LIN {X 0,Y 320.686,Z 443.971,A -85,B 0,C 180,E1 -15902.996,E2 -15902.996} C_VEL
LIN {X 0,Y 319.386,Z 457.296,A -85,B 0,C 180,E1 -15903.715,E2 -15903.715} C_VEL
LIN {X 0,Y 317.852,Z 469.93,A -85,B 0,C 180,E1 -15904.635,E2 -15904.635} C_VEL
LIN {X 0,Y 316.177,Z 481.923,A -85,B 0,C 180,E1 -15905.756,E2 -15905.756} C_VEL
LIN {X 0,Y 314.275,Z 493.762,A -85,B 0,C 180,E1 -15907.136,E2 -15907.136} C_VEL
LIN {X 0,Y 312.419,Z 503.822,A -85,B 0,C 180,E1 -15908.559,E2 -15908.559} C_VEL
LIN {X 0,Y 310.276,Z 514.883,A -85,B 0,C 180,E1 -15910.483,E2 -15910.483} C_VEL
LIN {X 0,Y 308.49,Z 524.011,A -85,B 0,C 180,E1 -15912.431,E2 -15912.431} C_VEL
LIN {X 0,Y 306.873,Z 532.736,A -85,B 0,C 180,E1 -15914.73,E2 -15914.73} C_VEL
LIN {X 0,Y 305.729,Z 538.879,A -85,B 0,C 180,E1 -15916.711,E2 -15916.711} C_VEL
LIN {X 0,Y 304.809,Z 543.968,A -85,B 0,C 180,E1 -15918.698,E2 -15918.698} C_VEL
LIN {X 0,Y 304.094,Z 549.221,A -85,B 0,C 180,E1 -15921.36,E2 -15921.36} C_VEL
LIN {X 0,Y 303.694,Z 553.281,A -85,B 0,C 180,E1 -15924.322,E2 -15924.322} C_VEL
LIN {X 0,Y 303.583,Z 554.856,A -85,B 0,C 180,E1 -15926.018,E2 -15926.018} C_VEL
LIN {X 0,Y 303.525,Z 556.187,A -85,B 0,C 180,E1 -15928.673,E2 -15928.673} C_VEL
LIN {X 0,Y 303.525,Z 556.181,A -85,B 0,C 180,E1 -15931.327,E2 -15931.327} C_VEL
LIN {X 0,Y 303.584,Z 554.841,A -85,B 0,C 180,E1 -15933.982,E2 -15933.982} C_VEL
LIN {X 0,Y 303.752,Z 552.139,A -85,B 0,C 180,E1 -15936.643,E2 -15936.643} C_VEL
LIN {X 0,Y 304.224,Z 548.001,A -85,B 0,C 180,E1 -15939.306,E2 -15939.306} C_VEL
LIN {X 0,Y 305.041,Z 542.303,A -85,B 0,C 180,E1 -15941.967,E2 -15941.967} C_VEL
LIN {X 0,Y 306.327,Z 535.882,A -85,B 0,C 180,E1 -15944.278,E2 -15944.278} C_VEL
LIN {X 0,Y 307.684,Z 527.905,A -85,B 0,C 180,E1 -15946.589,E2 -15946.589} C_VEL
LIN {X 0,Y 309.31,Z 519.557,A -85,B 0,C 180,E1 -15948.548,E2 -15948.548} C_VEL
LIN {X 0,Y 311.286,Z 509.51,A -85,B 0,C 180,E1 -15950.484,E2 -15950.484} C_VEL
LIN {X 0,Y 313.222,Z 499.398,A -85,B 0,C 180,E1 -15952.075,E2 -15952.075} C_VEL
LIN {X 0,Y 315.371,Z 487.142,A -85,B 0,C 180,E1 -15953.648,E2 -15953.648} C_VEL
LIN {X 0,Y 317.142,Z 474.986,A -85,B 0,C 180,E1 -15954.9,E2 -15954.9} C_VEL
LIN {X 0,Y 318.891,Z 461.491,A -85,B 0,C 180,E1 -15955.977,E2 -15955.977} C_VEL
LIN {X 0,Y 320.356,Z 447.369,A -85,B 0,C 180,E1 -15956.814,E2 -15956.814} C_VEL
LIN {X 0,Y 321.321,Z 433.529,A -85,B 0,C 180,E1 -15957.387,E2 -15957.387} C_VEL
LIN {X 0,Y 322.133,Z 414.857,A -85,B 0,C 180,E1 -15957.841,E2 -15957.841} C_VEL
LIN {X 0,Y 324.269,Z 337.737,A -85,B 0,C 180,E1 -15959.546,E2 -15959.546} C_VEL
LIN {X 0,Y 321.158,Z 321.063,A -85,B 0,C 180,E1 -15960.282,E2 -15960.282} C_VEL
LIN {X 0,Y 313.966,Z 304.498,A -85,B 0,C 180,E1 -15961.482,E2 -15961.482} C_VEL
LIN {X 0,Y 308.979,Z 293.727,A -85,B 0,C 180,E1 -15962.372,E2 -15962.372} C_VEL
LIN {X 0,Y 306.536,Z 284.268,A -85,B 0,C 180,E1 -15965.373,E2 -15965.373} C_VEL
LIN {X 0,Y 305.494,Z 280.07,A -85,B 0,C 180,E1 -15966.89,E2 -15966.89} C_VEL
LIN {X 0,Y 305.452,Z 280.04,A -85,B 0,C 180,E1 -15970.599,E2 -15970.599} C_VEL
LIN {X 0,Y 305.423,Z 280.062,A -85,B 0,C 180,E1 -15973.654,E2 -15973.654} C_VEL
LIN {X 0,Y 305.451,Z 280.062,A -85,B 0,C 180,E1 -15977.414,E2 -15977.414} C_VEL
LIN {X 0,Y 305.491,Z 280.058,A -85,B 0,C 180,E1 -15981.6,E2 -15981.6} C_VEL
LIN {X 0,Y 305.458,Z 280.011,A -85,B 0,C 180,E1 -15984.886,E2 -15984.886} C_VEL
LIN {X 0,Y 305.447,Z 280.048,A -85,B 0,C 180,E1 -15988.354,E2 -15988.354} C_VEL
LIN {X 0,Y 305.516,Z 280.05,A -85,B 0,C 180,E1 -15991.113,E2 -15991.113} C_VEL
LIN {X 0,Y 305.566,Z 280.043,A -85,B 0,C 180,E1 -15994.088,E2 -15994.088} C_VEL
LIN {X 0,Y 305.496,Z 280.042,A -85,B 0,C 180,E1 -15998.403,E2 -15998.403} C_VEL
LIN {X 0,Y 305.585,Z 280.045,A -85,B 0,C 180,E1 -16001.217,E2 -16001.217} C_VEL
LIN {X 0,Y 305.643,Z 280.032,A -85,B 0,C 180,E1 -16005.349,E2 -16005.349} C_VEL
LIN {X 0,Y 305.632,Z 280.02,A -85,B 0,C 180,E1 -16009.4,E2 -16009.4} C_VEL
LIN {X 0,Y 305.807,Z 280.017,A -85,B 0,C 180,E1 -16012.074,E2 -16012.074} C_VEL
LIN {X 0,Y 305.682,Z 280.021,A -85,B 0,C 180,E1 -16014.723,E2 -16014.723} C_VEL
LIN {X 0,Y 305.951,Z 279.997,A -85,B 0,C 180,E1 -16018.684,E2 -16018.684} C_VEL
LIN {X 0,Y 305.951,Z 279.983,A -85,B 0,C 180,E1 -16021.316,E2 -16021.316} C_VEL
LIN {X 0,Y 305.682,Z 280.033,A -85,B 0,C 180,E1 -16025.277,E2 -16025.277} C_VEL
LIN {X 0,Y 305.791,Z 280.004,A -85,B 0,C 180,E1 -16027.926,E2 -16027.926} C_VEL
LIN {X 0,Y 305.597,Z 280.042,A -85,B 0,C 180,E1 -16031.945,E2 -16031.945} C_VEL
LIN {X 0,Y 305.632,Z 280.021,A -85,B 0,C 180,E1 -16035.035,E2 -16035.035} C_VEL
LIN {X 0,Y 305.571,Z 280.038,A -85,B 0,C 180,E1 -16039.445,E2 -16039.445} C_VEL
LIN {X 0,Y 305.486,Z 280.056,A -85,B 0,C 180,E1 -16043.042,E2 -16043.042} C_VEL
LIN {X 0,Y 305.543,Z 280.034,A -85,B 0,C 180,E1 -16046.228,E2 -16046.228} C_VEL
LIN {X 0,Y 305.492,Z 280.058,A -85,B 0,C 180,E1 -16049.051,E2 -16049.051} C_VEL
LIN {X 0,Y 305.461,Z 280.007,A -85,B 0,C 180,E1 -16053.517,E2 -16053.517} C_VEL
LIN {X 0,Y 305.494,Z 280.05,A -85,B 0,C 180,E1 -16056.737,E2 -16056.737} C_VEL
LIN {X 0,Y 305.454,Z 280.025,A -85,B 0,C 180,E1 -16060.601,E2 -16060.601} C_VEL
LIN {X 0,Y 305.417,Z 280.065,A -85,B 0,C 180,E1 -16064.493,E2 -16064.493} C_VEL
LIN {X 0,Y 305.44,Z 280.038,A -85,B 0,C 180,E1 -16068.144,E2 -16068.144} C_VEL
LIN {X 0,Y 305.466,Z 280.045,A -85,B 0,C 180,E1 -16071.597,E2 -16071.597} C_VEL
LIN {X 0,Y 305.522,Z 280.246,A -85,B 0,C 180,E1 -16074.593,E2 -16074.593} C_VEL
LIN {X 0,Y 307.66,Z 288.77,A -85,B 0,C 180,E1 -16077.486,E2 -16077.486} C_VEL
LIN {X 0,Y 310.081,Z 293.827,A -85,B 0,C 180,E1 -16077.97,E2 -16077.97} C_VEL
LIN {X 0,Y 318.342,Z 311.367,A -85,B 0,C 180,E1 -16079.351,E2 -16079.351} C_VEL
LIN {X 0,Y 323.483,Z 324.294,A -85,B 0,C 180,E1 -16080.216,E2 -16080.216} C_VEL
LIN {X 0,Y 324.572,Z 329.961,A -85,B 0,C 180,E1 -16080.467,E2 -16080.467} C_VEL
LIN {X 0,Y 322.075,Z 413.055,A -85,B 0,C 180,E1 -16082.286,E2 -16082.286} C_VEL
LIN {X 0,Y 321.429,Z 429.29,A -85,B 0,C 180,E1 -16082.712,E2 -16082.712} C_VEL
LIN {X 0,Y 320.408,Z 442.749,A -85,B 0,C 180,E1 -16083.279,E2 -16083.279} C_VEL
LIN {X 0,Y 319.032,Z 456.662,A -85,B 0,C 180,E1 -16084.123,E2 -16084.123} C_VEL
LIN {X 0,Y 317.305,Z 470.455,A -85,B 0,C 180,E1 -16085.246,E2 -16085.246} C_VEL
LIN {X 0,Y 315.543,Z 482.714,A -85,B 0,C 180,E1 -16086.54,E2 -16086.54} C_VEL
LIN {X 0,Y 313.618,Z 493.673,A -85,B 0,C 180,E1 -16087.954,E2 -16087.954} C_VEL
LIN {X 0,Y 311.725,Z 503.803,A -85,B 0,C 180,E1 -16089.546,E2 -16089.546} C_VEL
LIN {X 0,Y 309.697,Z 513.859,A -85,B 0,C 180,E1 -16091.476,E2 -16091.476} C_VEL
LIN {X 0,Y 307.923,Z 523.001,A -85,B 0,C 180,E1 -16093.644,E2 -16093.644} C_VEL
LIN {X 0,Y 306.641,Z 530.178,A -85,B 0,C 180,E1 -16095.737,E2 -16095.737} C_VEL
LIN {X 0,Y 305.34,Z 536.596,A -85,B 0,C 180,E1 -16098.045,E2 -16098.045} C_VEL
LIN {X 0,Y 304.429,Z 542.285,A -85,B 0,C 180,E1 -16100.7,E2 -16100.7} C_VEL
LIN {X 0,Y 303.921,Z 546.419,A -85,B 0,C 180,E1 -16103.361,E2 -16103.361} C_VEL
LIN {X 0,Y 303.673,Z 549.122,A -85,B 0,C 180,E1 -16106.019,E2 -16106.019} C_VEL
LIN {X 0,Y 303.538,Z 550.476,A -85,B 0,C 180,E1 -16108.673,E2 -16108.673} C_VEL
LIN {X 0,Y 303.538,Z 550.507,A -85,B 0,C 180,E1 -16111.327,E2 -16111.327} C_VEL
LIN {X 0,Y 303.673,Z 549.213,A -85,B 0,C 180,E1 -16113.981,E2 -16113.981} C_VEL
LIN {X 0,Y 303.92,Z 546.564,A -85,B 0,C 180,E1 -16116.639,E2 -16116.639} C_VEL
LIN {X 0,Y 304.418,Z 542.492,A -85,B 0,C 180,E1 -16119.3,E2 -16119.3} C_VEL
LIN {X 0,Y 305.314,Z 536.866,A -85,B 0,C 180,E1 -16121.956,E2 -16121.956} C_VEL
LIN {X 0,Y 306.586,Z 530.512,A -85,B 0,C 180,E1 -16124.266,E2 -16124.266} C_VEL
LIN {X 0,Y 308.067,Z 522.382,A -85,B 0,C 180,E1 -16126.633,E2 -16126.633} C_VEL
LIN {X 0,Y 309.653,Z 514.35,A -85,B 0,C 180,E1 -16128.526,E2 -16128.526} C_VEL
LIN {X 0,Y 311.6,Z 504.392,A -85,B 0,C 180,E1 -16130.462,E2 -16130.462} C_VEL
LIN {X 0,Y 313.732,Z 493.305,A -85,B 0,C 180,E1 -16132.211,E2 -16132.211} C_VEL
LIN {X 0,Y 315.655,Z 482.266,A -85,B 0,C 180,E1 -16133.625,E2 -16133.625} C_VEL
LIN {X 0,Y 317.426,Z 470.279,A -85,B 0,C 180,E1 -16134.876,E2 -16134.876} C_VEL
LIN {X 0,Y 319.064,Z 457.023,A -85,B 0,C 180,E1 -16135.962,E2 -16135.962} C_VEL
LIN {X 0,Y 320.387,Z 443.995,A -85,B 0,C 180,E1 -16136.767,E2 -16136.767} C_VEL
LIN {X 0,Y 321.438,Z 429.999,A -85,B 0,C 180,E1 -16137.375,E2 -16137.375} C_VEL
LIN {X 0,Y 322.139,Z 412.365,A -85,B 0,C 180,E1 -16137.84,E2 -16137.84} C_VEL
LIN {X 0,Y 324.009,Z 350.719,A -85,B 0,C 180,E1 -16139.188,E2 -16139.188} C_VEL
LIN {X 0,Y 324.421,Z 329.108,A -85,B 0,C 180,E1 -16139.685,E2 -16139.685} C_VEL
LIN {X 0,Y 323.131,Z 323.106,A -85,B 0,C 180,E1 -16139.967,E2 -16139.967} C_VEL
LIN {X 0,Y 315.3,Z 304.632,A -85,B 0,C 180,E1 -16141.273,E2 -16141.273} C_VEL
LIN {X 0,Y 307.781,Z 289.059,A -85,B 0,C 180,E1 -16142.584,E2 -16142.584} C_VEL
LIN {X 0,Y 306.579,Z 284.524,A -85,B 0,C 180,E1 -16144.015,E2 -16144.015} C_VEL
LIN {X 0,Y 306.149,Z 282.788,A -85,B 0,C 180,E1 -16144.61,E2 -16144.61} C_VEL
LIN {X 0,Y 305.43,Z 281.38,A -85,B 0,C 180,E1 -16145.27,E2 -16145.27} C_VEL
LIN {X 0,Y 303.733,Z 280.518,A -85,B 0,C 180,E1 -16146.312,E2 -16146.312} C_VEL
LIN {X 0,Y 299.402,Z 280.805,A -85,B 0,C 180,E1 -16148.856,E2 -16148.856} C_VEL
LIN {X 0,Y 298.436,Z 280.938,A -85,B 0,C 180,E1 -16150.005,E2 -16150.005} C_VEL
LIN {X 0,Y 298.362,Z 280.932,A -85,B 0,C 180,E1 -16150.393,E2 -16150.393} C_VEL
LIN {X 0,Y 298.396,Z 280.916,A -85,B 0,C 180,E1 -16153.102,E2 -16153.102} C_VEL
LIN {X 0,Y 298.4,Z 280.916,A -85,B 0,C 180,E1 -16156.92,E2 -16156.92} C_VEL
LIN {X 0,Y 298.418,Z 280.931,A -85,B 0,C 180,E1 -16161.001,E2 -16161.001} C_VEL
LIN {X 0,Y 298.427,Z 280.925,A -85,B 0,C 180,E1 -16163.931,E2 -16163.931} C_VEL
LIN {X 0,Y 298.39,Z 280.899,A -85,B 0,C 180,E1 -16167.983,E2 -16167.983} C_VEL
LIN {X 0,Y 298.459,Z 280.933,A -85,B 0,C 180,E1 -16171.904,E2 -16171.904} C_VEL
LIN {X 0,Y 298.48,Z 280.92,A -85,B 0,C 180,E1 -16174.923,E2 -16174.923} C_VEL
LIN {X 0,Y 298.444,Z 280.918,A -85,B 0,C 180,E1 -16179.315,E2 -16179.315} C_VEL
LIN {X 0,Y 298.532,Z 280.923,A -85,B 0,C 180,E1 -16182.179,E2 -16182.179} C_VEL
LIN {X 0,Y 298.587,Z 280.898,A -85,B 0,C 180,E1 -16184.994,E2 -16184.994} C_VEL
LIN {X 0,Y 298.585,Z 280.911,A -85,B 0,C 180,E1 -16189.146,E2 -16189.146} C_VEL
LIN {X 0,Y 298.735,Z 280.88,A -85,B 0,C 180,E1 -16191.885,E2 -16191.885} C_VEL
LIN {X 0,Y 298.652,Z 280.91,A -85,B 0,C 180,E1 -16194.599,E2 -16194.599} C_VEL
LIN {X 0,Y 298.918,Z 280.858,A -85,B 0,C 180,E1 -16198.653,E2 -16198.653} C_VEL
LIN {X 0,Y 298.918,Z 280.873,A -85,B 0,C 180,E1 -16201.347,E2 -16201.347} C_VEL
LIN {X 0,Y 298.791,Z 280.892,A -85,B 0,C 180,E1 -16206.754,E2 -16206.754} C_VEL
LIN {X 0,Y 298.674,Z 280.89,A -85,B 0,C 180,E1 -16209.481,E2 -16209.481} C_VEL
LIN {X 0,Y 298.545,Z 280.922,A -85,B 0,C 180,E1 -16213.616,E2 -16213.616} C_VEL
LIN {X 0,Y 298.542,Z 280.904,A -85,B 0,C 180,E1 -16216.409,E2 -16216.409} C_VEL
LIN {X 0,Y 298.506,Z 280.927,A -85,B 0,C 180,E1 -16219.655,E2 -16219.655} C_VEL
LIN {X 0,Y 298.452,Z 280.927,A -85,B 0,C 180,E1 -16223.598,E2 -16223.598} C_VEL
LIN {X 0,Y 298.484,Z 280.918,A -85,B 0,C 180,E1 -16226.575,E2 -16226.575} C_VEL
LIN {X 0,Y 298.416,Z 280.938,A -85,B 0,C 180,E1 -16229.641,E2 -16229.641} C_VEL
LIN {X 0,Y 298.39,Z 280.903,A -85,B 0,C 180,E1 -16232.801,E2 -16232.801} C_VEL
LIN {X 0,Y 298.442,Z 280.913,A -85,B 0,C 180,E1 -16236.808,E2 -16236.808} C_VEL
LIN {X 0,Y 298.404,Z 280.935,A -85,B 0,C 180,E1 -16239.487,E2 -16239.487} C_VEL
LIN {X 0,Y 298.422,Z 280.935,A -85,B 0,C 180,E1 -16243.11,E2 -16243.11} C_VEL
LIN {X 0,Y 298.464,Z 280.915,A -85,B 0,C 180,E1 -16246.933,E2 -16246.933} C_VEL
LIN {X 0,Y 298.431,Z 280.937,A -85,B 0,C 180,E1 -16251,E2 -16251} C_VEL
LIN {X 0,Y 298.481,Z 280.971,A -85,B 0,C 180,E1 -16252.384,E2 -16252.384} C_VEL
LIN {X 0,Y 301.015,Z 291,A -85,B 0,C 180,E1 -16255.921,E2 -16255.921} C_VEL
LIN {X 0,Y 301.722,Z 293.772,A -85,B 0,C 180,E1 -16256.725,E2 -16256.725} C_VEL
LIN {X 0,Y 310.639,Z 312.674,A -85,B 0,C 180,E1 -16258.33,E2 -16258.33} C_VEL
LIN {X 0,Y 315.731,Z 325.016,A -85,B 0,C 180,E1 -16259.217,E2 -16259.217} C_VEL
LIN {X 0,Y 318.186,Z 339.496,A -85,B 0,C 180,E1 -16259.851,E2 -16259.851} C_VEL
LIN {X 0,Y 315.386,Z 429.211,A -85,B 0,C 180,E1 -16261.873,E2 -16261.873} C_VEL
LIN {X 0,Y 314.376,Z 443.915,A -85,B 0,C 180,E1 -16262.409,E2 -16262.409} C_VEL
LIN {X 0,Y 313.05,Z 457.237,A -85,B 0,C 180,E1 -16263.141,E2 -16263.141} C_VEL
LIN {X 0,Y 311.442,Z 469.869,A -85,B 0,C 180,E1 -16264.074,E2 -16264.074} C_VEL
LIN {X 0,Y 309.639,Z 482.266,A -85,B 0,C 180,E1 -16265.26,E2 -16265.26} C_VEL
LIN {X 0,Y 307.497,Z 494.874,A -85,B 0,C 180,E1 -16266.781,E2 -16266.781} C_VEL
LIN {X 0,Y 305.352,Z 505.724,A -85,B 0,C 180,E1 -16268.392,E2 -16268.392} C_VEL
LIN {X 0,Y 303.216,Z 516.448,A -85,B 0,C 180,E1 -16270.362,E2 -16270.362} C_VEL
LIN {X 0,Y 301.404,Z 525.302,A -85,B 0,C 180,E1 -16272.355,E2 -16272.355} C_VEL
LIN {X 0,Y 299.755,Z 533.789,A -85,B 0,C 180,E1 -16274.707,E2 -16274.707} C_VEL
LIN {X 0,Y 298.419,Z 540.627,A -85,B 0,C 180,E1 -16277.072,E2 -16277.072} C_VEL
LIN {X 0,Y 297.591,Z 545.338,A -85,B 0,C 180,E1 -16279.11,E2 -16279.11} C_VEL
LIN {X 0,Y 296.91,Z 550.222,A -85,B 0,C 180,E1 -16281.835,E2 -16281.835} C_VEL
LIN {X 0,Y 296.553,Z 553.616,A -85,B 0,C 180,E1 -16284.561,E2 -16284.561} C_VEL
LIN {X 0,Y 296.481,Z 555.623,A -85,B 0,C 180,E1 -16287.283,E2 -16287.283} C_VEL
LIN {X 0,Y 296.45,Z 556.284,A -85,B 0,C 180,E1 -16290,E2 -16290} C_VEL
LIN {X 0,Y 296.481,Z 555.612,A -85,B 0,C 180,E1 -16292.717,E2 -16292.717} C_VEL
LIN {X 0,Y 296.587,Z 553.433,A -85,B 0,C 180,E1 -16295.592,E2 -16295.592} C_VEL
LIN {X 0,Y 296.91,Z 550.189,A -85,B 0,C 180,E1 -16298.165,E2 -16298.165} C_VEL
LIN {X 0,Y 297.593,Z 545.288,A -85,B 0,C 180,E1 -16300.89,E2 -16300.89} C_VEL
LIN {X 0,Y 298.419,Z 540.563,A -85,B 0,C 180,E1 -16302.928,E2 -16302.928} C_VEL
LIN {X 0,Y 299.732,Z 533.725,A -85,B 0,C 180,E1 -16305.29,E2 -16305.29} C_VEL
LIN {X 0,Y 301.113,Z 526.564,A -85,B 0,C 180,E1 -16307.312,E2 -16307.312} C_VEL
LIN {X 0,Y 302.891,Z 517.962,A -85,B 0,C 180,E1 -16309.307,E2 -16309.307} C_VEL
LIN {X 0,Y 304.954,Z 507.536,A -85,B 0,C 180,E1 -16311.283,E2 -16311.283} C_VEL
LIN {X 0,Y 307.098,Z 497.053,A -85,B 0,C 180,E1 -16312.895,E2 -16312.895} C_VEL
LIN {X 0,Y 309.239,Z 484.476,A -85,B 0,C 180,E1 -16314.472,E2 -16314.472} C_VEL
LIN {X 0,Y 311.205,Z 471.378,A -85,B 0,C 180,E1 -16315.767,E2 -16315.767} C_VEL
LIN {X 0,Y 312.923,Z 458.027,A -85,B 0,C 180,E1 -16316.781,E2 -16316.781} C_VEL
LIN {X 0,Y 314.294,Z 444.238,A -85,B 0,C 180,E1 -16317.554,E2 -16317.554} C_VEL
LIN {X 0,Y 315.369,Z 429.817,A -85,B 0,C 180,E1 -16318.084,E2 -16318.084} C_VEL
LIN {X 0,Y 318.117,Z 339.637,A -85,B 0,C 180,E1 -16320.125,E2 -16320.125} C_VEL
LIN {X 0,Y 315.49,Z 324.243,A -85,B 0,C 180,E1 -16320.8,E2 -16320.8} C_VEL
LIN {X 0,Y 308.305,Z 307.631,A -85,B 0,C 180,E1 -16322.042,E2 -16322.042} C_VEL
LIN {X 0,Y 301.672,Z 293.605,A -85,B 0,C 180,E1 -16323.26,E2 -16323.26} C_VEL
LIN {X 0,Y 299.336,Z 284.508,A -85,B 0,C 180,E1 -16326.258,E2 -16326.258} C_VEL
LIN {X 0,Y 298.44,Z 280.947,A -85,B 0,C 180,E1 -16327.621,E2 -16327.621} C_VEL
LIN {X 0,Y 298.381,Z 280.915,A -85,B 0,C 180,E1 -16331.261,E2 -16331.261} C_VEL
LIN {X 0,Y 298.351,Z 280.943,A -85,B 0,C 180,E1 -16335.034,E2 -16335.034} C_VEL
LIN {X 0,Y 298.38,Z 280.934,A -85,B 0,C 180,E1 -16338.738,E2 -16338.738} C_VEL
LIN {X 0,Y 298.421,Z 280.932,A -85,B 0,C 180,E1 -16342.243,E2 -16342.243} C_VEL
LIN {X 0,Y 298.403,Z 280.887,A -85,B 0,C 180,E1 -16345.581,E2 -16345.581} C_VEL
LIN {X 0,Y 298.391,Z 280.934,A -85,B 0,C 180,E1 -16348.791,E2 -16348.791} C_VEL
LIN {X 0,Y 298.459,Z 280.92,A -85,B 0,C 180,E1 -16351.904,E2 -16351.904} C_VEL
LIN {X 0,Y 298.481,Z 280.929,A -85,B 0,C 180,E1 -16354.924,E2 -16354.924} C_VEL
LIN {X 0,Y 298.445,Z 280.928,A -85,B 0,C 180,E1 -16359.315,E2 -16359.315} C_VEL
LIN {X 0,Y 298.532,Z 280.913,A -85,B 0,C 180,E1 -16362.179,E2 -16362.179} C_VEL
LIN {X 0,Y 298.588,Z 280.909,A -85,B 0,C 180,E1 -16364.995,E2 -16364.995} C_VEL
LIN {X 0,Y 298.587,Z 280.898,A -85,B 0,C 180,E1 -16369.146,E2 -16369.146} C_VEL
LIN {X 0,Y 298.753,Z 280.893,A -85,B 0,C 180,E1 -16371.886,E2 -16371.886} C_VEL
LIN {X 0,Y 298.654,Z 280.898,A -85,B 0,C 180,E1 -16374.599,E2 -16374.599} C_VEL
LIN {X 0,Y 298.917,Z 280.873,A -85,B 0,C 180,E1 -16378.653,E2 -16378.653} C_VEL
LIN {X 0,Y 298.918,Z 280.859,A -85,B 0,C 180,E1 -16381.347,E2 -16381.347} C_VEL
LIN {X 0,Y 298.782,Z 280.89,A -85,B 0,C 180,E1 -16386.754,E2 -16386.754} C_VEL
LIN {X 0,Y 298.63,Z 280.893,A -85,B 0,C 180,E1 -16389.482,E2 -16389.482} C_VEL
LIN {X 0,Y 298.546,Z 280.911,A -85,B 0,C 180,E1 -16393.616,E2 -16393.616} C_VEL
LIN {X 0,Y 298.543,Z 280.914,A -85,B 0,C 180,E1 -16396.409,E2 -16396.409} C_VEL
LIN {X 0,Y 298.506,Z 280.917,A -85,B 0,C 180,E1 -16399.655,E2 -16399.655} C_VEL
LIN {X 0,Y 298.453,Z 280.934,A -85,B 0,C 180,E1 -16403.598,E2 -16403.598} C_VEL
LIN {X 0,Y 298.485,Z 280.914,A -85,B 0,C 180,E1 -16406.575,E2 -16406.575} C_VEL
LIN {X 0,Y 298.417,Z 280.935,A -85,B 0,C 180,E1 -16409.642,E2 -16409.642} C_VEL
LIN {X 0,Y 298.391,Z 280.889,A -85,B 0,C 180,E1 -16412.801,E2 -16412.801} C_VEL
LIN {X 0,Y 298.462,Z 280.926,A -85,B 0,C 180,E1 -16416.813,E2 -16416.813} C_VEL
LIN {X 0,Y 298.411,Z 280.92,A -85,B 0,C 180,E1 -16419.486,E2 -16419.486} C_VEL
LIN {X 0,Y 298.396,Z 280.913,A -85,B 0,C 180,E1 -16423.104,E2 -16423.104} C_VEL
LIN {X 0,Y 298.401,Z 280.916,A -85,B 0,C 180,E1 -16426.921,E2 -16426.921} C_VEL
LIN {X 0,Y 298.397,Z 280.932,A -85,B 0,C 180,E1 -16431.008,E2 -16431.008} C_VEL
LIN {X 0,Y 298.464,Z 281.067,A -85,B 0,C 180,E1 -16433.845,E2 -16433.845} C_VEL
LIN {X 0,Y 300.51,Z 288.901,A -85,B 0,C 180,E1 -16436.622,E2 -16436.622} C_VEL
LIN {X 0,Y 303.356,Z 294.889,A -85,B 0,C 180,E1 -16437.198,E2 -16437.198} C_VEL
LIN {X 0,Y 311.058,Z 310.831,A -85,B 0,C 180,E1 -16438.535,E2 -16438.535} C_VEL
LIN {X 0,Y 317.44,Z 326.268,A -85,B 0,C 180,E1 -16439.638,E2 -16439.638} C_VEL
LIN {X 0,Y 318.353,Z 331.68,A -85,B 0,C 180,E1 -16439.873,E2 -16439.873} C_VEL
LIN {X 0,Y 315.887,Z 411.357,A -85,B 0,C 180,E1 -16441.65,E2 -16441.65} C_VEL
LIN {X 0,Y 315.155,Z 429.372,A -85,B 0,C 180,E1 -16442.122,E2 -16442.122} C_VEL
LIN {X 0,Y 314.028,Z 443.587,A -85,B 0,C 180,E1 -16442.736,E2 -16442.736} C_VEL
LIN {X 0,Y 312.642,Z 456.736,A -85,B 0,C 180,E1 -16443.553,E2 -16443.553} C_VEL
LIN {X 0,Y 310.879,Z 470.492,A -85,B 0,C 180,E1 -16444.695,E2 -16444.695} C_VEL
LIN {X 0,Y 309.042,Z 482.785,A -85,B 0,C 180,E1 -16446.015,E2 -16446.015} C_VEL
LIN {X 0,Y 306.824,Z 494.811,A -85,B 0,C 180,E1 -16447.617,E2 -16447.617} C_VEL
LIN {X 0,Y 304.695,Z 505.652,A -85,B 0,C 180,E1 -16449.406,E2 -16449.406} C_VEL
LIN {X 0,Y 302.639,Z 515.411,A -85,B 0,C 180,E1 -16451.379,E2 -16451.379} C_VEL
LIN {X 0,Y 300.993,Z 523.541,A -85,B 0,C 180,E1 -16453.391,E2 -16453.391} C_VEL
LIN {X 0,Y 299.753,Z 530.246,A -85,B 0,C 180,E1 -16455.402,E2 -16455.402} C_VEL
LIN {X 0,Y 298.355,Z 536.664,A -85,B 0,C 180,E1 -16457.76,E2 -16457.76} C_VEL
LIN {X 0,Y 297.39,Z 542.353,A -85,B 0,C 180,E1 -16460.478,E2 -16460.478} C_VEL
LIN {X 0,Y 296.854,Z 546.486,A -85,B 0,C 180,E1 -16463.202,E2 -16463.202} C_VEL
LIN {X 0,Y 296.575,Z 549.189,A -85,B 0,C 180,E1 -16465.923,E2 -16465.923} C_VEL
LIN {X 0,Y 296.46,Z 550.542,A -85,B 0,C 180,E1 -16468.642,E2 -16468.642} C_VEL
LIN {X 0,Y 296.459,Z 550.573,A -85,B 0,C 180,E1 -16471.358,E2 -16471.358} C_VEL
LIN {X 0,Y 296.575,Z 549.279,A -85,B 0,C 180,E1 -16474.077,E2 -16474.077} C_VEL
LIN {X 0,Y 296.854,Z 546.63,A -85,B 0,C 180,E1 -16476.798,E2 -16476.798} C_VEL
LIN {X 0,Y 297.377,Z 542.557,A -85,B 0,C 180,E1 -16479.522,E2 -16479.522} C_VEL
LIN {X 0,Y 298.329,Z 536.932,A -85,B 0,C 180,E1 -16482.24,E2 -16482.24} C_VEL
LIN {X 0,Y 299.696,Z 530.577,A -85,B 0,C 180,E1 -16484.601,E2 -16484.601} C_VEL
LIN {X 0,Y 301.114,Z 522.987,A -85,B 0,C 180,E1 -16486.875,E2 -16486.875} C_VEL
LIN {X 0,Y 302.893,Z 514.414,A -85,B 0,C 180,E1 -16488.955,E2 -16488.955} C_VEL
LIN {X 0,Y 304.93,Z 504.456,A -85,B 0,C 180,E1 -16490.93,E2 -16490.93} C_VEL
LIN {X 0,Y 307.17,Z 493.368,A -85,B 0,C 180,E1 -16492.711,E2 -16492.711} C_VEL
LIN {X 0,Y 309.171,Z 482.327,A -85,B 0,C 180,E1 -16494.152,E2 -16494.152} C_VEL
LIN {X 0,Y 310.976,Z 470.34,A -85,B 0,C 180,E1 -16495.429,E2 -16495.429} C_VEL
LIN {X 0,Y 312.701,Z 457.082,A -85,B 0,C 180,E1 -16496.531,E2 -16496.531} C_VEL
LIN {X 0,Y 314.07,Z 444.051,A -85,B 0,C 180,E1 -16497.35,E2 -16497.35} C_VEL
LIN {X 0,Y 315.166,Z 430.049,A -85,B 0,C 180,E1 -16497.968,E2 -16497.968} C_VEL
LIN {X 0,Y 315.894,Z 412.407,A -85,B 0,C 180,E1 -16498.44,E2 -16498.44} C_VEL
LIN {X 0,Y 317.784,Z 353.431,A -85,B 0,C 180,E1 -16499.748,E2 -16499.748} C_VEL
LIN {X 0,Y 318.334,Z 330.709,A -85,B 0,C 180,E1 -16500.272,E2 -16500.272} C_VEL
LIN {X 0,Y 317.386,Z 326.064,A -85,B 0,C 180,E1 -16500.491,E2 -16500.491} C_VEL
LIN {X 0,Y 309.604,Z 307.643,A -85,B 0,C 180,E1 -16501.836,E2 -16501.836} C_VEL
LIN {X 0,Y 302.014,Z 292.202,A -85,B 0,C 180,E1 -16503.165,E2 -16503.165} C_VEL
LIN {X 0,Y 300.432,Z 288.707,A -85,B 0,C 180,E1 -16503.545,E2 -16503.545} C_VEL
LIN {X 0,Y 298.47,Z 281.117,A -85,B 0,C 180,E1 -16506.246,E2 -16506.246} C_VEL
LIN {X 0,Y 298.399,Z 280.939,A -85,B 0,C 180,E1 -16509.487,E2 -16509.487} C_VEL
LIN {X 0,Y 298.362,Z 280.932,A -85,B 0,C 180,E1 -16510.393,E2 -16510.393} C_VEL
LIN {X 0,Y 297.71,Z 281.012,A -85,B 0,C 180,E1 -16511.52,E2 -16511.52} C_VEL
LIN {X 0,Y 294.888,Z 281.378,A -85,B 0,C 180,E1 -16513.356,E2 -16513.356} C_VEL
LIN {X 0,Y 292.472,Z 281.684,A -85,B 0,C 180,E1 -16514.845,E2 -16514.845} C_VEL
LIN {X 0,Y 291.413,Z 281.805,A -85,B 0,C 180,E1 -16515.999,E2 -16515.999} C_VEL
LIN {X 0,Y 291.315,Z 281.808,A -85,B 0,C 180,E1 -16516.39,E2 -16516.39} C_VEL
LIN {X 0,Y 291.388,Z 281.793,A -85,B 0,C 180,E1 -16520.515,E2 -16520.515} C_VEL
LIN {X 0,Y 291.422,Z 281.812,A -85,B 0,C 180,E1 -16522.922,E2 -16522.922} C_VEL
LIN {X 0,Y 291.34,Z 281.768,A -85,B 0,C 180,E1 -16526.301,E2 -16526.301} C_VEL
LIN {X 0,Y 291.383,Z 281.812,A -85,B 0,C 180,E1 -16530.259,E2 -16530.259} C_VEL
LIN {X 0,Y 291.411,Z 281.795,A -85,B 0,C 180,E1 -16534.271,E2 -16534.271} C_VEL
LIN {X 0,Y 291.376,Z 281.812,A -85,B 0,C 180,E1 -16537.299,E2 -16537.299} C_VEL
LIN {X 0,Y 291.453,Z 281.794,A -85,B 0,C 180,E1 -16540.27,E2 -16540.27} C_VEL
LIN {X 0,Y 291.535,Z 281.777,A -85,B 0,C 180,E1 -16544.634,E2 -16544.634} C_VEL
LIN {X 0,Y 291.529,Z 281.792,A -85,B 0,C 180,E1 -16548.88,E2 -16548.88} C_VEL
LIN {X 0,Y 291.681,Z 281.757,A -85,B 0,C 180,E1 -16551.688,E2 -16551.688} C_VEL
LIN {X 0,Y 291.622,Z 281.786,A -85,B 0,C 180,E1 -16554.468,E2 -16554.468} C_VEL
LIN {X 0,Y 291.884,Z 281.733,A -85,B 0,C 180,E1 -16558.62,E2 -16558.62} C_VEL
LIN {X 0,Y 291.884,Z 281.749,A -85,B 0,C 180,E1 -16561.38,E2 -16561.38} C_VEL
LIN {X 0,Y 291.739,Z 281.769,A -85,B 0,C 180,E1 -16566.918,E2 -16566.918} C_VEL
LIN {X 0,Y 291.623,Z 281.766,A -85,B 0,C 180,E1 -16569.712,E2 -16569.712} C_VEL
LIN {X 0,Y 291.515,Z 281.799,A -85,B 0,C 180,E1 -16573.951,E2 -16573.951} C_VEL
LIN {X 0,Y 291.481,Z 281.784,A -85,B 0,C 180,E1 -16576.818,E2 -16576.818} C_VEL
LIN {X 0,Y 291.445,Z 281.807,A -85,B 0,C 180,E1 -16579.875,E2 -16579.875} C_VEL
LIN {X 0,Y 291.395,Z 281.811,A -85,B 0,C 180,E1 -16584.206,E2 -16584.206} C_VEL
LIN {X 0,Y 291.417,Z 281.795,A -85,B 0,C 180,E1 -16587.272,E2 -16587.272} C_VEL
LIN {X 0,Y 291.333,Z 281.819,A -85,B 0,C 180,E1 -16590.437,E2 -16590.437} C_VEL
LIN {X 0,Y 291.339,Z 281.769,A -85,B 0,C 180,E1 -16593.699,E2 -16593.699} C_VEL
LIN {X 0,Y 291.377,Z 281.803,A -85,B 0,C 180,E1 -16597.256,E2 -16597.256} C_VEL
LIN {X 0,Y 291.333,Z 281.809,A -85,B 0,C 180,E1 -16600.642,E2 -16600.642} C_VEL
LIN {X 0,Y 291.338,Z 281.813,A -85,B 0,C 180,E1 -16604.393,E2 -16604.393} C_VEL
LIN {X 0,Y 291.385,Z 281.785,A -85,B 0,C 180,E1 -16608.391,E2 -16608.391} C_VEL
LIN {X 0,Y 291.425,Z 281.927,A -85,B 0,C 180,E1 -16611.68,E2 -16611.68} C_VEL
LIN {X 0,Y 293.777,Z 290.926,A -85,B 0,C 180,E1 -16614.961,E2 -16614.961} C_VEL
LIN {X 0,Y 294.451,Z 293.564,A -85,B 0,C 180,E1 -16615.781,E2 -16615.781} C_VEL
LIN {X 0,Y 303.669,Z 312.839,A -85,B 0,C 180,E1 -16617.521,E2 -16617.521} C_VEL
LIN {X 0,Y 309.857,Z 327.379,A -85,B 0,C 180,E1 -16618.632,E2 -16618.632} C_VEL
LIN {X 0,Y 312.063,Z 340.503,A -85,B 0,C 180,E1 -16619.223,E2 -16619.223} C_VEL
LIN {X 0,Y 309.158,Z 429.163,A -85,B 0,C 180,E1 -16621.254,E2 -16621.254} C_VEL
LIN {X 0,Y 308.114,Z 443.858,A -85,B 0,C 180,E1 -16621.798,E2 -16621.798} C_VEL
LIN {X 0,Y 306.742,Z 457.177,A -85,B 0,C 180,E1 -16622.543,E2 -16622.543} C_VEL
LIN {X 0,Y 305.071,Z 469.808,A -85,B 0,C 180,E1 -16623.491,E2 -16623.491} C_VEL
LIN {X 0,Y 303.061,Z 482.921,A -85,B 0,C 180,E1 -16624.778,E2 -16624.778} C_VEL
LIN {X 0,Y 300.963,Z 494.81,A -85,B 0,C 180,E1 -16626.246,E2 -16626.246} C_VEL
LIN {X 0,Y 298.74,Z 505.66,A -85,B 0,C 180,E1 -16627.889,E2 -16627.889} C_VEL
LIN {X 0,Y 296.498,Z 516.383,A -85,B 0,C 180,E1 -16629.898,E2 -16629.898} C_VEL
LIN {X 0,Y 294.609,Z 525.237,A -85,B 0,C 180,E1 -16631.934,E2 -16631.934} C_VEL
LIN {X 0,Y 292.888,Z 533.723,A -85,B 0,C 180,E1 -16634.339,E2 -16634.339} C_VEL
LIN {X 0,Y 291.476,Z 540.561,A -85,B 0,C 180,E1 -16636.759,E2 -16636.759} C_VEL
LIN {X 0,Y 290.578,Z 545.272,A -85,B 0,C 180,E1 -16638.844,E2 -16638.844} C_VEL
LIN {X 0,Y 289.86,Z 550.156,A -85,B 0,C 180,E1 -16641.635,E2 -16641.635} C_VEL
LIN {X 0,Y 289.471,Z 553.646,A -85,B 0,C 180,E1 -16644.519,E2 -16644.519} C_VEL
LIN {X 0,Y 289.388,Z 555.557,A -85,B 0,C 180,E1 -16647.216,E2 -16647.216} C_VEL
LIN {X 0,Y 289.37,Z 556.218,A -85,B 0,C 180,E1 -16650,E2 -16650} C_VEL
LIN {X 0,Y 289.388,Z 555.545,A -85,B 0,C 180,E1 -16652.784,E2 -16652.784} C_VEL
LIN {X 0,Y 289.48,Z 553.529,A -85,B 0,C 180,E1 -16655.573,E2 -16655.573} C_VEL
LIN {X 0,Y 289.86,Z 550.121,A -85,B 0,C 180,E1 -16658.365,E2 -16658.365} C_VEL
LIN {X 0,Y 290.58,Z 545.22,A -85,B 0,C 180,E1 -16661.156,E2 -16661.156} C_VEL
LIN {X 0,Y 291.476,Z 540.495,A -85,B 0,C 180,E1 -16663.242,E2 -16663.242} C_VEL
LIN {X 0,Y 292.851,Z 533.672,A -85,B 0,C 180,E1 -16665.654,E2 -16665.654} C_VEL
LIN {X 0,Y 294.298,Z 526.494,A -85,B 0,C 180,E1 -16667.726,E2 -16667.726} C_VEL
LIN {X 0,Y 296.169,Z 517.892,A -85,B 0,C 180,E1 -16669.764,E2 -16669.764} C_VEL
LIN {X 0,Y 298.32,Z 507.466,A -85,B 0,C 180,E1 -16671.78,E2 -16671.78} C_VEL
LIN {X 0,Y 300.563,Z 496.983,A -85,B 0,C 180,E1 -16673.422,E2 -16673.422} C_VEL
LIN {X 0,Y 302.752,Z 484.405,A -85,B 0,C 180,E1 -16675.031,E2 -16675.031} C_VEL
LIN {X 0,Y 304.817,Z 471.306,A -85,B 0,C 180,E1 -16676.348,E2 -16676.348} C_VEL
LIN {X 0,Y 306.587,Z 457.954,A -85,B 0,C 180,E1 -16677.38,E2 -16677.38} C_VEL
LIN {X 0,Y 308.022,Z 444.162,A -85,B 0,C 180,E1 -16678.165,E2 -16678.165} C_VEL
LIN {X 0,Y 309.124,Z 429.733,A -85,B 0,C 180,E1 -16678.703,E2 -16678.703} C_VEL
LIN {X 0,Y 311.924,Z 342.841,A -85,B 0,C 180,E1 -16680.701,E2 -16680.701} C_VEL
LIN {X 0,Y 311.599,Z 338.261,A -85,B 0,C 180,E1 -16680.857,E2 -16680.857} C_VEL
LIN {X 0,Y 309.484,Z 326.458,A -85,B 0,C 180,E1 -16681.404,E2 -16681.404} C_VEL
LIN {X 0,Y 301.76,Z 308.636,A -85,B 0,C 180,E1 -16682.793,E2 -16682.793} C_VEL
LIN {X 0,Y 295.598,Z 296.169,A -85,B 0,C 180,E1 -16683.92,E2 -16683.92} C_VEL
LIN {X 0,Y 294.347,Z 293.248,A -85,B 0,C 180,E1 -16684.25,E2 -16684.25} C_VEL
LIN {X 0,Y 291.989,Z 284.154,A -85,B 0,C 180,E1 -16687.412,E2 -16687.412} C_VEL
LIN {X 0,Y 291.363,Z 281.836,A -85,B 0,C 180,E1 -16688.376,E2 -16688.376} C_VEL
LIN {X 0,Y 291.316,Z 281.798,A -85,B 0,C 180,E1 -16692.492,E2 -16692.492} C_VEL
LIN {X 0,Y 291.306,Z 281.817,A -85,B 0,C 180,E1 -16696.366,E2 -16696.366} C_VEL
LIN {X 0,Y 291.383,Z 281.81,A -85,B 0,C 180,E1 -16700.516,E2 -16700.516} C_VEL
LIN {X 0,Y 291.407,Z 281.792,A -85,B 0,C 180,E1 -16702.92,E2 -16702.92} C_VEL
LIN {X 0,Y 291.34,Z 281.769,A -85,B 0,C 180,E1 -16706.301,E2 -16706.301} C_VEL
LIN {X 0,Y 291.383,Z 281.814,A -85,B 0,C 180,E1 -16710.26,E2 -16710.26} C_VEL
LIN {X 0,Y 291.413,Z 281.808,A -85,B 0,C 180,E1 -16714.272,E2 -16714.272} C_VEL
LIN {X 0,Y 291.377,Z 281.799,A -85,B 0,C 180,E1 -16717.299,E2 -16717.299} C_VEL
LIN {X 0,Y 291.453,Z 281.806,A -85,B 0,C 180,E1 -16720.27,E2 -16720.27} C_VEL
LIN {X 0,Y 291.535,Z 281.783,A -85,B 0,C 180,E1 -16724.634,E2 -16724.634} C_VEL
LIN {X 0,Y 291.531,Z 281.779,A -85,B 0,C 180,E1 -16728.88,E2 -16728.88} C_VEL
LIN {X 0,Y 291.703,Z 281.768,A -85,B 0,C 180,E1 -16731.688,E2 -16731.688} C_VEL
LIN {X 0,Y 291.624,Z 281.775,A -85,B 0,C 180,E1 -16734.468,E2 -16734.468} C_VEL
LIN {X 0,Y 291.884,Z 281.749,A -85,B 0,C 180,E1 -16738.62,E2 -16738.62} C_VEL
LIN {X 0,Y 291.884,Z 281.734,A -85,B 0,C 180,E1 -16741.38,E2 -16741.38} C_VEL
LIN {X 0,Y 291.73,Z 281.765,A -85,B 0,C 180,E1 -16746.918,E2 -16746.918} C_VEL
LIN {X 0,Y 291.569,Z 281.773,A -85,B 0,C 180,E1 -16749.714,E2 -16749.714} C_VEL
LIN {X 0,Y 291.516,Z 281.784,A -85,B 0,C 180,E1 -16753.951,E2 -16753.951} C_VEL
LIN {X 0,Y 291.482,Z 281.795,A -85,B 0,C 180,E1 -16756.818,E2 -16756.818} C_VEL
LIN {X 0,Y 291.446,Z 281.794,A -85,B 0,C 180,E1 -16759.875,E2 -16759.875} C_VEL
LIN {X 0,Y 291.396,Z 281.812,A -85,B 0,C 180,E1 -16764.206,E2 -16764.206} C_VEL
LIN {X 0,Y 291.419,Z 281.799,A -85,B 0,C 180,E1 -16767.272,E2 -16767.272} C_VEL
LIN {X 0,Y 291.334,Z 281.807,A -85,B 0,C 180,E1 -16770.437,E2 -16770.437} C_VEL
LIN {X 0,Y 291.341,Z 281.764,A -85,B 0,C 180,E1 -16773.699,E2 -16773.699} C_VEL
LIN {X 0,Y 291.396,Z 281.812,A -85,B 0,C 180,E1 -16777.26,E2 -16777.26} C_VEL
LIN {X 0,Y 291.334,Z 281.782,A -85,B 0,C 180,E1 -16780.643,E2 -16780.643} C_VEL
LIN {X 0,Y 291.313,Z 281.821,A -85,B 0,C 180,E1 -16784.398,E2 -16784.398} C_VEL
LIN {X 0,Y 291.325,Z 281.797,A -85,B 0,C 180,E1 -16788.405,E2 -16788.405} C_VEL
LIN {X 0,Y 291.346,Z 281.808,A -85,B 0,C 180,E1 -16791.158,E2 -16791.158} C_VEL
LIN {X 0,Y 291.449,Z 282.002,A -85,B 0,C 180,E1 -16793.143,E2 -16793.143} C_VEL
LIN {X 0,Y 293.301,Z 289.109,A -85,B 0,C 180,E1 -16795.709,E2 -16795.709} C_VEL
LIN {X 0,Y 302.351,Z 307.249,A -85,B 0,C 180,E1 -16797.417,E2 -16797.417} C_VEL
LIN {X 0,Y 309.242,Z 322.926,A -85,B 0,C 180,E1 -16798.652,E2 -16798.652} C_VEL
LIN {X 0,Y 311.745,Z 329.377,A -85,B 0,C 180,E1 -16799.102,E2 -16799.102} C_VEL
LIN {X 0,Y 312.22,Z 332.956,A -85,B 0,C 180,E1 -16799.249,E2 -16799.249} C_VEL
LIN {X 0,Y 309.612,Z 413.236,A -85,B 0,C 180,E1 -16801.068,E2 -16801.068} C_VEL
LIN {X 0,Y 308.828,Z 430.592,A -85,B 0,C 180,E1 -16801.545,E2 -16801.545} C_VEL
LIN {X 0,Y 307.679,Z 444.425,A -85,B 0,C 180,E1 -16802.172,E2 -16802.172} C_VEL
LIN {X 0,Y 306.193,Z 457.934,A -85,B 0,C 180,E1 -16803.044,E2 -16803.044} C_VEL
LIN {X 0,Y 304.429,Z 470.894,A -85,B 0,C 180,E1 -16804.157,E2 -16804.157} C_VEL
LIN {X 0,Y 302.563,Z 482.856,A -85,B 0,C 180,E1 -16805.468,E2 -16805.468} C_VEL
LIN {X 0,Y 300.269,Z 494.881,A -85,B 0,C 180,E1 -16807.101,E2 -16807.101} C_VEL
LIN {X 0,Y 298.039,Z 505.722,A -85,B 0,C 180,E1 -16808.924,E2 -16808.924} C_VEL
LIN {X 0,Y 295.886,Z 515.48,A -85,B 0,C 180,E1 -16810.938,E2 -16810.938} C_VEL
LIN {X 0,Y 294.281,Z 522.924,A -85,B 0,C 180,E1 -16812.8,E2 -16812.8} C_VEL
LIN {X 0,Y 292.881,Z 530.315,A -85,B 0,C 180,E1 -16815.051,E2 -16815.051} C_VEL
LIN {X 0,Y 291.384,Z 536.732,A -85,B 0,C 180,E1 -16817.463,E2 -16817.463} C_VEL
LIN {X 0,Y 290.364,Z 542.421,A -85,B 0,C 180,E1 -16820.246,E2 -16820.246} C_VEL
LIN {X 0,Y 289.775,Z 546.554,A -85,B 0,C 180,E1 -16823.035,E2 -16823.035} C_VEL
LIN {X 0,Y 289.482,Z 549.256,A -85,B 0,C 180,E1 -16825.823,E2 -16825.823} C_VEL
LIN {X 0,Y 289.384,Z 550.609,A -85,B 0,C 180,E1 -16828.608,E2 -16828.608} C_VEL
LIN {X 0,Y 289.384,Z 550.64,A -85,B 0,C 180,E1 -16831.392,E2 -16831.392} C_VEL
LIN {X 0,Y 289.482,Z 549.345,A -85,B 0,C 180,E1 -16834.177,E2 -16834.177} C_VEL
LIN {X 0,Y 289.775,Z 546.696,A -85,B 0,C 180,E1 -16836.965,E2 -16836.965} C_VEL
LIN {X 0,Y 290.349,Z 542.623,A -85,B 0,C 180,E1 -16839.755,E2 -16839.755} C_VEL
LIN {X 0,Y 291.357,Z 536.997,A -85,B 0,C 180,E1 -16842.538,E2 -16842.538} C_VEL
LIN {X 0,Y 292.81,Z 530.642,A -85,B 0,C 180,E1 -16844.952,E2 -16844.952} C_VEL
LIN {X 0,Y 294.399,Z 522.675,A -85,B 0,C 180,E1 -16847.381,E2 -16847.381} C_VEL
LIN {X 0,Y 296.164,Z 514.478,A -85,B 0,C 180,E1 -16849.403,E2 -16849.403} C_VEL
LIN {X 0,Y 298.299,Z 504.519,A -85,B 0,C 180,E1 -16851.418,E2 -16851.418} C_VEL
LIN {X 0,Y 300.626,Z 493.431,A -85,B 0,C 180,E1 -16853.234,E2 -16853.234} C_VEL
LIN {X 0,Y 302.711,Z 482.389,A -85,B 0,C 180,E1 -16854.702,E2 -16854.702} C_VEL
LIN {X 0,Y 304.573,Z 470.401,A -85,B 0,C 180,E1 -16856.003,E2 -16856.003} C_VEL
LIN {X 0,Y 306.37,Z 457.141,A -85,B 0,C 180,E1 -16857.124,E2 -16857.124} C_VEL
LIN {X 0,Y 307.782,Z 444.107,A -85,B 0,C 180,E1 -16857.957,E2 -16857.957} C_VEL
LIN {X 0,Y 308.928,Z 430.1,A -85,B 0,C 180,E1 -16858.584,E2 -16858.584} C_VEL
LIN {X 0,Y 309.683,Z 412.449,A -85,B 0,C 180,E1 -16859.064,E2 -16859.064} C_VEL
LIN {X 0,Y 311.652,Z 353.473,A -85,B 0,C 180,E1 -16860.395,E2 -16860.395} C_VEL
LIN {X 0,Y 312.142,Z 331.431,A -85,B 0,C 180,E1 -16860.92,E2 -16860.92} C_VEL
LIN {X 0,Y 311.399,Z 328.325,A -85,B 0,C 180,E1 -16861.084,E2 -16861.084} C_VEL
LIN {X 0,Y 303.937,Z 310.687,A -85,B 0,C 180,E1 -16862.419,E2 -16862.419} C_VEL
LIN {X 0,Y 296.949,Z 296.339,A -85,B 0,C 180,E1 -16863.689,E2 -16863.689} C_VEL
LIN {X 0,Y 293.275,Z 289.091,A -85,B 0,C 180,E1 -16864.424,E2 -16864.424} C_VEL
LIN {X 0,Y 291.426,Z 282.049,A -85,B 0,C 180,E1 -16866.968,E2 -16866.968} C_VEL
LIN {X 0,Y 291.346,Z 281.807,A -85,B 0,C 180,E1 -16868.842,E2 -16868.842} C_VEL
LIN {X 0,Y 291.317,Z 281.795,A -85,B 0,C 180,E1 -16872.492,E2 -16872.492} C_VEL
LIN {X 0,Y 291.315,Z 281.808,A -85,B 0,C 180,E1 -16876.39,E2 -16876.39} C_VEL
LIN {X 0,Y 290.628,Z 281.88,A -85,B 0,C 180,E1 -16877.543,E2 -16877.543} C_VEL
LIN {X 0,Y 287.814,Z 282.244,A -85,B 0,C 180,E1 -16879.424,E2 -16879.424} C_VEL
LIN {X 0,Y 285.439,Z 282.557,A -85,B 0,C 180,E1 -16880.95,E2 -16880.95} C_VEL
LIN {X 0,Y 284.413,Z 282.686,A -85,B 0,C 180,E1 -16882.132,E2 -16882.132} C_VEL
LIN {X 0,Y 284.325,Z 282.694,A -85,B 0,C 180,E1 -16882.532,E2 -16882.532} C_VEL
LIN {X 0,Y 284.319,Z 282.65,A -85,B 0,C 180,E1 -16885.352,E2 -16885.352} C_VEL
LIN {X 0,Y 284.291,Z 282.665,A -85,B 0,C 180,E1 -16888.725,E2 -16888.725} C_VEL
LIN {X 0,Y 284.393,Z 282.675,A -85,B 0,C 180,E1 -16892.826,E2 -16892.826} C_VEL
LIN {X 0,Y 284.361,Z 282.691,A -85,B 0,C 180,E1 -16896.706,E2 -16896.706} C_VEL
LIN {X 0,Y 284.398,Z 282.682,A -85,B 0,C 180,E1 -16901.261,E2 -16901.261} C_VEL
LIN {X 0,Y 284.472,Z 282.657,A -85,B 0,C 180,E1 -16904.469,E2 -16904.469} C_VEL
LIN {X 0,Y 284.481,Z 282.673,A -85,B 0,C 180,E1 -16908.601,E2 -16908.601} C_VEL
LIN {X 0,Y 284.633,Z 282.634,A -85,B 0,C 180,E1 -16911.48,E2 -16911.48} C_VEL
LIN {X 0,Y 284.592,Z 282.661,A -85,B 0,C 180,E1 -16914.331,E2 -16914.331} C_VEL
LIN {X 0,Y 284.85,Z 282.609,A -85,B 0,C 180,E1 -16918.586,E2 -16918.586} C_VEL
LIN {X 0,Y 284.85,Z 282.626,A -85,B 0,C 180,E1 -16921.414,E2 -16921.414} C_VEL
LIN {X 0,Y 284.692,Z 282.647,A -85,B 0,C 180,E1 -16927.09,E2 -16927.09} C_VEL
LIN {X 0,Y 284.56,Z 282.644,A -85,B 0,C 180,E1 -16929.955,E2 -16929.955} C_VEL
LIN {X 0,Y 284.472,Z 282.672,A -85,B 0,C 180,E1 -16934.303,E2 -16934.303} C_VEL
LIN {X 0,Y 284.419,Z 282.666,A -85,B 0,C 180,E1 -16937.249,E2 -16937.249} C_VEL
LIN {X 0,Y 284.373,Z 282.683,A -85,B 0,C 180,E1 -16940.243,E2 -16940.243} C_VEL
LIN {X 0,Y 284.364,Z 282.683,A -85,B 0,C 180,E1 -16943.876,E2 -16943.876} C_VEL
LIN {X 0,Y 284.392,Z 282.669,A -85,B 0,C 180,E1 -16947.174,E2 -16947.174} C_VEL
LIN {X 0,Y 284.291,Z 282.687,A -85,B 0,C 180,E1 -16951.275,E2 -16951.275} C_VEL
LIN {X 0,Y 284.336,Z 282.642,A -85,B 0,C 180,E1 -16955.349,E2 -16955.349} C_VEL
LIN {X 0,Y 284.314,Z 282.695,A -85,B 0,C 180,E1 -16958.169,E2 -16958.169} C_VEL
LIN {X 0,Y 284.283,Z 282.7,A -85,B 0,C 180,E1 -16962.129,E2 -16962.129} C_VEL
LIN {X 0,Y 284.316,Z 282.69,A -85,B 0,C 180,E1 -16966.202,E2 -16966.202} C_VEL
LIN {X 0,Y 284.362,Z 282.683,A -85,B 0,C 180,E1 -16970.476,E2 -16970.476} C_VEL
LIN {X 0,Y 284.379,Z 282.919,A -85,B 0,C 180,E1 -16970.937,E2 -16970.937} C_VEL
LIN {X 0,Y 286.553,Z 291.131,A -85,B 0,C 180,E1 -16974.033,E2 -16974.033} C_VEL
LIN {X 0,Y 287.192,Z 293.473,A -85,B 0,C 180,E1 -16974.789,E2 -16974.789} C_VEL
LIN {X 0,Y 295.171,Z 309.683,A -85,B 0,C 180,E1 -16976.376,E2 -16976.376} C_VEL
LIN {X 0,Y 303.011,Z 327.338,A -85,B 0,C 180,E1 -16977.84,E2 -16977.84} C_VEL
LIN {X 0,Y 304.121,Z 330.34,A -85,B 0,C 180,E1 -16978.053,E2 -16978.053} C_VEL
LIN {X 0,Y 305.946,Z 342.052,A -85,B 0,C 180,E1 -16978.581,E2 -16978.581} C_VEL
LIN {X 0,Y 302.966,Z 429.114,A -85,B 0,C 180,E1 -16980.61,E2 -16980.61} C_VEL
LIN {X 0,Y 301.878,Z 443.801,A -85,B 0,C 180,E1 -16981.162,E2 -16981.162} C_VEL
LIN {X 0,Y 300.468,Z 457.118,A -85,B 0,C 180,E1 -16981.919,E2 -16981.919} C_VEL
LIN {X 0,Y 298.729,Z 469.747,A -85,B 0,C 180,E1 -16982.883,E2 -16982.883} C_VEL
LIN {X 0,Y 296.584,Z 483.104,A -85,B 0,C 180,E1 -16984.219,E2 -16984.219} C_VEL
LIN {X 0,Y 294.455,Z 494.747,A -85,B 0,C 180,E1 -16985.688,E2 -16985.688} C_VEL
LIN {X 0,Y 292.156,Z 505.596,A -85,B 0,C 180,E1 -16987.364,E2 -16987.364} C_VEL
LIN {X 0,Y 289.817,Z 516.319,A -85,B 0,C 180,E1 -16989.414,E2 -16989.414} C_VEL
LIN {X 0,Y 287.81,Z 525.172,A -85,B 0,C 180,E1 -16991.492,E2 -16991.492} C_VEL
LIN {X 0,Y 286.233,Z 532.72,A -85,B 0,C 180,E1 -16993.658,E2 -16993.658} C_VEL
LIN {X 0,Y 284.964,Z 538.682,A -85,B 0,C 180,E1 -16995.722,E2 -16995.722} C_VEL
LIN {X 0,Y 283.808,Z 543.771,A -85,B 0,C 180,E1 -16997.849,E2 -16997.849} C_VEL
LIN {X 0,Y 282.946,Z 549.022,A -85,B 0,C 180,E1 -17000.709,E2 -17000.709} C_VEL
LIN {X 0,Y 282.572,Z 551.965,A -85,B 0,C 180,E1 -17002.857,E2 -17002.857} C_VEL
LIN {X 0,Y 282.304,Z 554.657,A -85,B 0,C 180,E1 -17005.717,E2 -17005.717} C_VEL
LIN {X 0,Y 282.295,Z 555.988,A -85,B 0,C 180,E1 -17008.574,E2 -17008.574} C_VEL
LIN {X 0,Y 282.295,Z 555.982,A -85,B 0,C 180,E1 -17011.427,E2 -17011.427} C_VEL
LIN {X 0,Y 282.304,Z 554.639,A -85,B 0,C 180,E1 -17014.283,E2 -17014.283} C_VEL
LIN {X 0,Y 282.572,Z 551.937,A -85,B 0,C 180,E1 -17017.144,E2 -17017.144} C_VEL
LIN {X 0,Y 283.126,Z 547.797,A -85,B 0,C 180,E1 -17020.006,E2 -17020.006} C_VEL
LIN {X 0,Y 284.132,Z 542.098,A -85,B 0,C 180,E1 -17022.862,E2 -17022.862} C_VEL
LIN {X 0,Y 285.52,Z 535.676,A -85,B 0,C 180,E1 -17025.343,E2 -17025.343} C_VEL
LIN {X 0,Y 287.195,Z 527.696,A -85,B 0,C 180,E1 -17027.811,E2 -17027.811} C_VEL
LIN {X 0,Y 289.104,Z 519.35,A -85,B 0,C 180,E1 -17029.897,E2 -17029.897} C_VEL
LIN {X 0,Y 291.32,Z 509.301,A -85,B 0,C 180,E1 -17031.958,E2 -17031.958} C_VEL
LIN {X 0,Y 293.793,Z 498.086,A -85,B 0,C 180,E1 -17033.808,E2 -17033.808} C_VEL
LIN {X 0,Y 295.914,Z 486.929,A -85,B 0,C 180,E1 -17035.309,E2 -17035.309} C_VEL
LIN {X 0,Y 297.933,Z 474.77,A -85,B 0,C 180,E1 -17036.627,E2 -17036.627} C_VEL
LIN {X 0,Y 299.865,Z 461.271,A -85,B 0,C 180,E1 -17037.762,E2 -17037.762} C_VEL
LIN {X 0,Y 301.494,Z 447.143,A -85,B 0,C 180,E1 -17038.641,E2 -17038.641} C_VEL
LIN {X 0,Y 302.608,Z 433.29,A -85,B 0,C 180,E1 -17039.238,E2 -17039.238} C_VEL
LIN {X 0,Y 303.62,Z 411.016,A -85,B 0,C 180,E1 -17039.797,E2 -17039.797} C_VEL
LIN {X 0,Y 305.79,Z 340.996,A -85,B 0,C 180,E1 -17041.434,E2 -17041.434} C_VEL
LIN {X 0,Y 303.737,Z 329.345,A -85,B 0,C 180,E1 -17041.987,E2 -17041.987} C_VEL
LIN {X 0,Y 297.241,Z 314.15,A -85,B 0,C 180,E1 -17043.198,E2 -17043.198} C_VEL
LIN {X 0,Y 290.431,Z 300.066,A -85,B 0,C 180,E1 -17044.491,E2 -17044.491} C_VEL
LIN {X 0,Y 287.138,Z 293.312,A -85,B 0,C 180,E1 -17045.203,E2 -17045.203} C_VEL
LIN {X 0,Y 284.631,Z 284.103,A -85,B 0,C 180,E1 -17048.542,E2 -17048.542} C_VEL
LIN {X 0,Y 284.325,Z 282.723,A -85,B 0,C 180,E1 -17049.186,E2 -17049.186} C_VEL
LIN {X 0,Y 284.266,Z 282.673,A -85,B 0,C 180,E1 -17052.124,E2 -17052.124} C_VEL
LIN {X 0,Y 284.252,Z 282.695,A -85,B 0,C 180,E1 -17056.189,E2 -17056.189} C_VEL
LIN {X 0,Y 284.304,Z 282.687,A -85,B 0,C 180,E1 -17060.023,E2 -17060.023} C_VEL
LIN {X 0,Y 284.33,Z 282.657,A -85,B 0,C 180,E1 -17063.614,E2 -17063.614} C_VEL
LIN {X 0,Y 284.304,Z 282.656,A -85,B 0,C 180,E1 -17067.189,E2 -17067.189} C_VEL
LIN {X 0,Y 284.355,Z 282.689,A -85,B 0,C 180,E1 -17070.376,E2 -17070.376} C_VEL
LIN {X 0,Y 284.374,Z 282.677,A -85,B 0,C 180,E1 -17073.586,E2 -17073.586} C_VEL
LIN {X 0,Y 284.362,Z 282.678,A -85,B 0,C 180,E1 -17076.707,E2 -17076.707} C_VEL
LIN {X 0,Y 284.399,Z 282.684,A -85,B 0,C 180,E1 -17081.261,E2 -17081.261} C_VEL
LIN {X 0,Y 284.473,Z 282.661,A -85,B 0,C 180,E1 -17084.47,E2 -17084.47} C_VEL
LIN {X 0,Y 284.483,Z 282.659,A -85,B 0,C 180,E1 -17088.601,E2 -17088.601} C_VEL
LIN {X 0,Y 284.654,Z 282.644,A -85,B 0,C 180,E1 -17091.481,E2 -17091.481} C_VEL
LIN {X 0,Y 284.595,Z 282.651,A -85,B 0,C 180,E1 -17094.331,E2 -17094.331} C_VEL
LIN {X 0,Y 284.85,Z 282.626,A -85,B 0,C 180,E1 -17098.586,E2 -17098.586} C_VEL
LIN {X 0,Y 284.85,Z 282.609,A -85,B 0,C 180,E1 -17101.414,E2 -17101.414} C_VEL
LIN {X 0,Y 284.681,Z 282.64,A -85,B 0,C 180,E1 -17107.091,E2 -17107.091} C_VEL
LIN {X 0,Y 284.514,Z 282.654,A -85,B 0,C 180,E1 -17109.957,E2 -17109.957} C_VEL
LIN {X 0,Y 284.473,Z 282.658,A -85,B 0,C 180,E1 -17114.303,E2 -17114.303} C_VEL
LIN {X 0,Y 284.42,Z 282.679,A -85,B 0,C 180,E1 -17117.249,E2 -17117.249} C_VEL
LIN {X 0,Y 284.374,Z 282.671,A -85,B 0,C 180,E1 -17120.243,E2 -17120.243} C_VEL
LIN {X 0,Y 284.365,Z 282.688,A -85,B 0,C 180,E1 -17123.876,E2 -17123.876} C_VEL
LIN {X 0,Y 284.393,Z 282.672,A -85,B 0,C 180,E1 -17127.174,E2 -17127.174} C_VEL
LIN {X 0,Y 284.292,Z 282.666,A -85,B 0,C 180,E1 -17131.275,E2 -17131.275} C_VEL
LIN {X 0,Y 284.358,Z 282.651,A -85,B 0,C 180,E1 -17135.355,E2 -17135.355} C_VEL
LIN {X 0,Y 284.326,Z 282.694,A -85,B 0,C 180,E1 -17138.167,E2 -17138.167} C_VEL
LIN {X 0,Y 284.267,Z 282.659,A -85,B 0,C 180,E1 -17142.125,E2 -17142.125} C_VEL
LIN {X 0,Y 284.267,Z 282.684,A -85,B 0,C 180,E1 -17146.193,E2 -17146.193} C_VEL
LIN {X 0,Y 284.305,Z 282.697,A -85,B 0,C 180,E1 -17150.025,E2 -17150.025} C_VEL
LIN {X 0,Y 284.318,Z 282.8,A -85,B 0,C 180,E1 -17152.28,E2 -17152.28} C_VEL
LIN {X 0,Y 286.058,Z 289.016,A -85,B 0,C 180,E1 -17154.682,E2 -17154.682} C_VEL
LIN {X 0,Y 288.529,Z 293.999,A -85,B 0,C 180,E1 -17155.247,E2 -17155.247} C_VEL
LIN {X 0,Y 297.147,Z 311.221,A -85,B 0,C 180,E1 -17156.884,E2 -17156.884} C_VEL
LIN {X 0,Y 303.772,Z 326.43,A -85,B 0,C 180,E1 -17158.114,E2 -17158.114} C_VEL
LIN {X 0,Y 306.029,Z 332.72,A -85,B 0,C 180,E1 -17158.548,E2 -17158.548} C_VEL
LIN {X 0,Y 304.005,Z 397.748,A -85,B 0,C 180,E1 -17160.067,E2 -17160.067} C_VEL
LIN {X 0,Y 302.944,Z 426.154,A -85,B 0,C 180,E1 -17160.752,E2 -17160.752} C_VEL
LIN {X 0,Y 301.771,Z 440.696,A -85,B 0,C 180,E1 -17161.341,E2 -17161.341} C_VEL
LIN {X 0,Y 300.283,Z 454.627,A -85,B 0,C 180,E1 -17162.185,E2 -17162.185} C_VEL
LIN {X 0,Y 298.569,Z 467.585,A -85,B 0,C 180,E1 -17163.245,E2 -17163.245} C_VEL
LIN {X 0,Y 296.597,Z 480.051,A -85,B 0,C 180,E1 -17164.554,E2 -17164.554} C_VEL
LIN {X 0,Y 294.403,Z 491.588,A -85,B 0,C 180,E1 -17166.058,E2 -17166.058} C_VEL
LIN {X 0,Y 292.185,Z 502.095,A -85,B 0,C 180,E1 -17167.739,E2 -17167.739} C_VEL
LIN {X 0,Y 289.915,Z 512.528,A -85,B 0,C 180,E1 -17169.792,E2 -17169.792} C_VEL
LIN {X 0,Y 287.89,Z 521.208,A -85,B 0,C 180,E1 -17171.886,E2 -17171.886} C_VEL
LIN {X 0,Y 286.248,Z 529.376,A -85,B 0,C 180,E1 -17174.332,E2 -17174.332} C_VEL
LIN {X 0,Y 284.822,Z 535.125,A -85,B 0,C 180,E1 -17176.443,E2 -17176.443} C_VEL
LIN {X 0,Y 283.856,Z 539.848,A -85,B 0,C 180,E1 -17178.576,E2 -17178.576} C_VEL
LIN {X 0,Y 282.967,Z 544.741,A -85,B 0,C 180,E1 -17181.43,E2 -17181.43} C_VEL
LIN {X 0,Y 282.523,Z 548.145,A -85,B 0,C 180,E1 -17184.289,E2 -17184.289} C_VEL
LIN {X 0,Y 282.357,Z 550.165,A -85,B 0,C 180,E1 -17187.147,E2 -17187.147} C_VEL
LIN {X 0,Y 282.296,Z 550.856,A -85,B 0,C 180,E1 -17190,E2 -17190} C_VEL
LIN {X 0,Y 282.357,Z 550.225,A -85,B 0,C 180,E1 -17192.853,E2 -17192.853} C_VEL
LIN {X 0,Y 282.559,Z 548.185,A -85,B 0,C 180,E1 -17195.782,E2 -17195.782} C_VEL
LIN {X 0,Y 282.965,Z 544.91,A -85,B 0,C 180,E1 -17198.57,E2 -17198.57} C_VEL
LIN {X 0,Y 283.825,Z 540.08,A -85,B 0,C 180,E1 -17201.425,E2 -17201.425} C_VEL
LIN {X 0,Y 284.793,Z 535.418,A -85,B 0,C 180,E1 -17203.558,E2 -17203.558} C_VEL
LIN {X 0,Y 286.351,Z 528.637,A -85,B 0,C 180,E1 -17206.028,E2 -17206.028} C_VEL
LIN {X 0,Y 288.144,Z 520.216,A -85,B 0,C 180,E1 -17208.486,E2 -17208.486} C_VEL
LIN {X 0,Y 290.2,Z 511.424,A -85,B 0,C 180,E1 -17210.558,E2 -17210.558} C_VEL
LIN {X 0,Y 292.513,Z 500.771,A -85,B 0,C 180,E1 -17212.607,E2 -17212.607} C_VEL
LIN {X 0,Y 294.799,Z 489.993,A -85,B 0,C 180,E1 -17214.282,E2 -17214.282} C_VEL
LIN {X 0,Y 297.002,Z 478.017,A -85,B 0,C 180,E1 -17215.797,E2 -17215.797} C_VEL
LIN {X 0,Y 298.944,Z 465.181,A -85,B 0,C 180,E1 -17217.096,E2 -17217.096} C_VEL
LIN {X 0,Y 300.737,Z 451.502,A -85,B 0,C 180,E1 -17218.148,E2 -17218.148} C_VEL
LIN {X 0,Y 302.23,Z 436.981,A -85,B 0,C 180,E1 -17218.944,E2 -17218.944} C_VEL
LIN {X 0,Y 303.142,Z 422.575,A -85,B 0,C 180,E1 -17219.467,E2 -17219.467} C_VEL
LIN {X 0,Y 305.433,Z 357.242,A -85,B 0,C 180,E1 -17220.981,E2 -17220.981} C_VEL
LIN {X 0,Y 306.075,Z 332.616,A -85,B 0,C 180,E1 -17221.571,E2 -17221.571} C_VEL
LIN {X 0,Y 300.894,Z 319.503,A -85,B 0,C 180,E1 -17222.544,E2 -17222.544} C_VEL
LIN {X 0,Y 292.302,Z 301.159,A -85,B 0,C 180,E1 -17224.159,E2 -17224.159} C_VEL
LIN {X 0,Y 286.061,Z 289.13,A -85,B 0,C 180,E1 -17225.426,E2 -17225.426} C_VEL
LIN {X 0,Y 284.361,Z 282.993,A -85,B 0,C 180,E1 -17227.732,E2 -17227.732} C_VEL
LIN {X 0,Y 284.296,Z 282.68,A -85,B 0,C 180,E1 -17228.17,E2 -17228.17} C_VEL
LIN {X 0,Y 284.266,Z 282.674,A -85,B 0,C 180,E1 -17232.123,E2 -17232.123} C_VEL
LIN {X 0,Y 284.255,Z 282.686,A -85,B 0,C 180,E1 -17236.374,E2 -17236.374} C_VEL
LIN {X 0,Y 284.305,Z 282.665,A -85,B 0,C 180,E1 -17240.023,E2 -17240.023} C_VEL
LIN {X 0,Y 284.325,Z 282.694,A -85,B 0,C 180,E1 -17242.532,E2 -17242.532} C_VEL
LIN {X 0,Y 283.632,Z 282.77,A -85,B 0,C 180,E1 -17243.714,E2 -17243.714} C_VEL
LIN {X 0,Y 280.742,Z 283.098,A -85,B 0,C 180,E1 -17245.64,E2 -17245.64} C_VEL
LIN {X 0,Y 278.316,Z 283.392,A -85,B 0,C 180,E1 -17247.205,E2 -17247.205} C_VEL
LIN {X 0,Y 277.298,Z 283.529,A -85,B 0,C 180,E1 -17248.418,E2 -17248.418} C_VEL
LIN {X 0,Y 277.228,Z 283.545,A -85,B 0,C 180,E1 -17248.829,E2 -17248.829} C_VEL
LIN {X 0,Y 277.354,Z 283.551,A -85,B 0,C 180,E1 -17252.863,E2 -17252.863} C_VEL
LIN {X 0,Y 277.324,Z 283.565,A -85,B 0,C 180,E1 -17256.079,E2 -17256.079} C_VEL
LIN {X 0,Y 277.34,Z 283.555,A -85,B 0,C 180,E1 -17260.766,E2 -17260.766} C_VEL
LIN {X 0,Y 277.422,Z 283.533,A -85,B 0,C 180,E1 -17265.325,E2 -17265.325} C_VEL
LIN {X 0,Y 277.455,Z 283.537,A -85,B 0,C 180,E1 -17269.787,E2 -17269.787} C_VEL
LIN {X 0,Y 277.635,Z 283.515,A -85,B 0,C 180,E1 -17272.728,E2 -17272.728} C_VEL
LIN {X 0,Y 277.816,Z 283.484,A -85,B 0,C 180,E1 -17278.55,E2 -17278.55} C_VEL
LIN {X 0,Y 277.816,Z 283.502,A -85,B 0,C 180,E1 -17281.449,E2 -17281.449} C_VEL
LIN {X 0,Y 277.646,Z 283.524,A -85,B 0,C 180,E1 -17287.271,E2 -17287.271} C_VEL
LIN {X 0,Y 277.501,Z 283.522,A -85,B 0,C 180,E1 -17290.211,E2 -17290.211} C_VEL
LIN {X 0,Y 277.422,Z 283.547,A -85,B 0,C 180,E1 -17294.675,E2 -17294.675} C_VEL
LIN {X 0,Y 277.34,Z 283.563,A -85,B 0,C 180,E1 -17299.234,E2 -17299.234} C_VEL
LIN {X 0,Y 277.314,Z 283.564,A -85,B 0,C 180,E1 -17304.171,E2 -17304.171} C_VEL
LIN {X 0,Y 277.321,Z 283.55,A -85,B 0,C 180,E1 -17307.506,E2 -17307.506} C_VEL
LIN {X 0,Y 277.267,Z 283.571,A -85,B 0,C 180,E1 -17310.482,E2 -17310.482} C_VEL
LIN {X 0,Y 277.242,Z 283.521,A -85,B 0,C 180,E1 -17313.896,E2 -17313.896} C_VEL
LIN {X 0,Y 277.268,Z 283.563,A -85,B 0,C 180,E1 -17317.469,E2 -17317.469} C_VEL
LIN {X 0,Y 277.214,Z 283.57,A -85,B 0,C 180,E1 -17321.236,E2 -17321.236} C_VEL
LIN {X 0,Y 277.244,Z 283.574,A -85,B 0,C 180,E1 -17325.218,E2 -17325.218} C_VEL
LIN {X 0,Y 277.292,Z 283.546,A -85,B 0,C 180,E1 -17329.495,E2 -17329.495} C_VEL
LIN {X 0,Y 277.367,Z 283.904,A -85,B 0,C 180,E1 -17330.144,E2 -17330.144} C_VEL
LIN {X 0,Y 279.703,Z 292.628,A -85,B 0,C 180,E1 -17333.519,E2 -17333.519} C_VEL
LIN {X 0,Y 279.941,Z 293.423,A -85,B 0,C 180,E1 -17333.736,E2 -17333.736} C_VEL
LIN {X 0,Y 287.035,Z 307.425,A -85,B 0,C 180,E1 -17335.224,E2 -17335.224} C_VEL
LIN {X 0,Y 295.553,Z 325.976,A -85,B 0,C 180,E1 -17336.889,E2 -17336.889} C_VEL
LIN {X 0,Y 298.308,Z 332.913,A -85,B 0,C 180,E1 -17337.427,E2 -17337.427} C_VEL
LIN {X 0,Y 299.891,Z 342.95,A -85,B 0,C 180,E1 -17337.898,E2 -17337.898} C_VEL
LIN {X 0,Y 296.818,Z 429.065,A -85,B 0,C 180,E1 -17339.939,E2 -17339.939} C_VEL
LIN {X 0,Y 295.679,Z 443.745,A -85,B 0,C 180,E1 -17340.498,E2 -17340.498} C_VEL
LIN {X 0,Y 294.214,Z 457.058,A -85,B 0,C 180,E1 -17341.267,E2 -17341.267} C_VEL
LIN {X 0,Y 292.434,Z 469.685,A -85,B 0,C 180,E1 -17342.249,E2 -17342.249} C_VEL
LIN {X 0,Y 290.209,Z 482.947,A -85,B 0,C 180,E1 -17343.597,E2 -17343.597} C_VEL
LIN {X 0,Y 287.99,Z 494.684,A -85,B 0,C 180,E1 -17345.105,E2 -17345.105} C_VEL
LIN {X 0,Y 285.594,Z 505.532,A -85,B 0,C 180,E1 -17346.814,E2 -17346.814} C_VEL
LIN {X 0,Y 283.159,Z 516.255,A -85,B 0,C 180,E1 -17348.907,E2 -17348.907} C_VEL
LIN {X 0,Y 281.05,Z 525.107,A -85,B 0,C 180,E1 -17351.03,E2 -17351.03} C_VEL
LIN {X 0,Y 279.231,Z 533.371,A -85,B 0,C 180,E1 -17353.477,E2 -17353.477} C_VEL
LIN {X 0,Y 277.62,Z 540.43,A -85,B 0,C 180,E1 -17356.085,E2 -17356.085} C_VEL
LIN {X 0,Y 276.544,Z 545.14,A -85,B 0,C 180,E1 -17358.27,E2 -17358.27} C_VEL
LIN {X 0,Y 275.76,Z 550.024,A -85,B 0,C 180,E1 -17361.204,E2 -17361.204} C_VEL
LIN {X 0,Y 275.301,Z 553.418,A -85,B 0,C 180,E1 -17364.139,E2 -17364.139} C_VEL
LIN {X 0,Y 275.21,Z 555.424,A -85,B 0,C 180,E1 -17367.073,E2 -17367.073} C_VEL
LIN {X 0,Y 275.218,Z 556.085,A -85,B 0,C 180,E1 -17370,E2 -17370} C_VEL
LIN {X 0,Y 275.21,Z 555.411,A -85,B 0,C 180,E1 -17372.928,E2 -17372.928} C_VEL
LIN {X 0,Y 275.335,Z 553.395,A -85,B 0,C 180,E1 -17375.86,E2 -17375.86} C_VEL
LIN {X 0,Y 275.761,Z 549.986,A -85,B 0,C 180,E1 -17378.796,E2 -17378.796} C_VEL
LIN {X 0,Y 276.545,Z 545.084,A -85,B 0,C 180,E1 -17381.73,E2 -17381.73} C_VEL
LIN {X 0,Y 278.057,Z 538.546,A -85,B 0,C 180,E1 -17384.64,E2 -17384.64} C_VEL
LIN {X 0,Y 279.527,Z 531.294,A -85,B 0,C 180,E1 -17387.174,E2 -17387.174} C_VEL
LIN {X 0,Y 281.683,Z 522.255,A -85,B 0,C 180,E1 -17389.683,E2 -17389.683} C_VEL
LIN {X 0,Y 283.927,Z 512.799,A -85,B 0,C 180,E1 -17391.795,E2 -17391.795} C_VEL
LIN {X 0,Y 286.316,Z 502.329,A -85,B 0,C 180,E1 -17393.699,E2 -17393.699} C_VEL
LIN {X 0,Y 288.777,Z 490.775,A -85,B 0,C 180,E1 -17395.4,E2 -17395.4} C_VEL
LIN {X 0,Y 290.766,Z 479.537,A -85,B 0,C 180,E1 -17396.754,E2 -17396.754} C_VEL
LIN {X 0,Y 292.722,Z 467.403,A -85,B 0,C 180,E1 -17397.916,E2 -17397.916} C_VEL
LIN {X 0,Y 294.551,Z 454.054,A -85,B 0,C 180,E1 -17398.892,E2 -17398.892} C_VEL
LIN {X 0,Y 295.979,Z 439.485,A -85,B 0,C 180,E1 -17399.665,E2 -17399.665} C_VEL
LIN {X 0,Y 296.961,Z 425.051,A -85,B 0,C 180,E1 -17400.143,E2 -17400.143} C_VEL
LIN {X 0,Y 299.78,Z 343.359,A -85,B 0,C 180,E1 -17402.071,E2 -17402.071} C_VEL
LIN {X 0,Y 298.143,Z 332.461,A -85,B 0,C 180,E1 -17402.572,E2 -17402.572} C_VEL
LIN {X 0,Y 292.273,Z 318.569,A -85,B 0,C 180,E1 -17403.708,E2 -17403.708} C_VEL
LIN {X 0,Y 284.067,Z 301.422,A -85,B 0,C 180,E1 -17405.334,E2 -17405.334} C_VEL
LIN {X 0,Y 279.885,Z 293.243,A -85,B 0,C 180,E1 -17406.254,E2 -17406.254} C_VEL
LIN {X 0,Y 277.348,Z 284.054,A -85,B 0,C 180,E1 -17409.744,E2 -17409.744} C_VEL
LIN {X 0,Y 277.263,Z 283.563,A -85,B 0,C 180,E1 -17410.198,E2 -17410.198} C_VEL
LIN {X 0,Y 277.207,Z 283.564,A -85,B 0,C 180,E1 -17413.197,E2 -17413.197} C_VEL
LIN {X 0,Y 277.212,Z 283.58,A -85,B 0,C 180,E1 -17417.325,E2 -17417.325} C_VEL
LIN {X 0,Y 277.267,Z 283.572,A -85,B 0,C 180,E1 -17421.79,E2 -17421.79} C_VEL
LIN {X 0,Y 277.281,Z 283.521,A -85,B 0,C 180,E1 -17424.341,E2 -17424.341} C_VEL
LIN {X 0,Y 277.241,Z 283.547,A -85,B 0,C 180,E1 -17427.836,E2 -17427.836} C_VEL
LIN {X 0,Y 277.285,Z 283.563,A -85,B 0,C 180,E1 -17431.212,E2 -17431.212} C_VEL
LIN {X 0,Y 277.31,Z 283.567,A -85,B 0,C 180,E1 -17434.479,E2 -17434.479} C_VEL
LIN {X 0,Y 277.281,Z 283.553,A -85,B 0,C 180,E1 -17437.654,E2 -17437.654} C_VEL
LIN {X 0,Y 277.34,Z 283.563,A -85,B 0,C 180,E1 -17440.766,E2 -17440.766} C_VEL
LIN {X 0,Y 277.423,Z 283.547,A -85,B 0,C 180,E1 -17445.325,E2 -17445.325} C_VEL
LIN {X 0,Y 277.501,Z 283.522,A -85,B 0,C 180,E1 -17449.789,E2 -17449.789} C_VEL
LIN {X 0,Y 277.647,Z 283.524,A -85,B 0,C 180,E1 -17452.729,E2 -17452.729} C_VEL
LIN {X 0,Y 277.816,Z 283.502,A -85,B 0,C 180,E1 -17458.551,E2 -17458.551} C_VEL
LIN {X 0,Y 277.816,Z 283.484,A -85,B 0,C 180,E1 -17461.45,E2 -17461.45} C_VEL
LIN {X 0,Y 277.635,Z 283.515,A -85,B 0,C 180,E1 -17467.271,E2 -17467.271} C_VEL
LIN {X 0,Y 277.456,Z 283.536,A -85,B 0,C 180,E1 -17470.213,E2 -17470.213} C_VEL
LIN {X 0,Y 277.423,Z 283.533,A -85,B 0,C 180,E1 -17474.675,E2 -17474.675} C_VEL
LIN {X 0,Y 277.341,Z 283.556,A -85,B 0,C 180,E1 -17479.234,E2 -17479.234} C_VEL
LIN {X 0,Y 277.315,Z 283.566,A -85,B 0,C 180,E1 -17484.171,E2 -17484.171} C_VEL
LIN {X 0,Y 277.322,Z 283.556,A -85,B 0,C 180,E1 -17487.506,E2 -17487.506} C_VEL
LIN {X 0,Y 277.269,Z 283.557,A -85,B 0,C 180,E1 -17490.482,E2 -17490.482} C_VEL
LIN {X 0,Y 277.251,Z 283.517,A -85,B 0,C 180,E1 -17493.895,E2 -17493.895} C_VEL
LIN {X 0,Y 277.283,Z 283.572,A -85,B 0,C 180,E1 -17497.467,E2 -17497.467} C_VEL
LIN {X 0,Y 277.208,Z 283.536,A -85,B 0,C 180,E1 -17501.237,E2 -17501.237} C_VEL
LIN {X 0,Y 277.215,Z 283.579,A -85,B 0,C 180,E1 -17505.224,E2 -17505.224} C_VEL
LIN {X 0,Y 277.22,Z 283.567,A -85,B 0,C 180,E1 -17509.513,E2 -17509.513} C_VEL
LIN {X 0,Y 277.263,Z 283.703,A -85,B 0,C 180,E1 -17511.453,E2 -17511.453} C_VEL
LIN {X 0,Y 278.85,Z 289.204,A -85,B 0,C 180,E1 -17513.646,E2 -17513.646} C_VEL
LIN {X 0,Y 286.11,Z 303.237,A -85,B 0,C 180,E1 -17515.186,E2 -17515.186} C_VEL
LIN {X 0,Y 293.292,Z 318.105,A -85,B 0,C 180,E1 -17516.588,E2 -17516.588} C_VEL
LIN {X 0,Y 298.9,Z 331.438,A -85,B 0,C 180,E1 -17517.669,E2 -17517.669} C_VEL
LIN {X 0,Y 300.009,Z 334.3,A -85,B 0,C 180,E1 -17517.883,E2 -17517.883} C_VEL
LIN {X 0,Y 297.525,Z 407.465,A -85,B 0,C 180,E1 -17519.61,E2 -17519.61} C_VEL
LIN {X 0,Y 296.629,Z 428.479,A -85,B 0,C 180,E1 -17520.163,E2 -17520.163} C_VEL
LIN {X 0,Y 295.433,Z 442.295,A -85,B 0,C 180,E1 -17520.764,E2 -17520.764} C_VEL
LIN {X 0,Y 293.878,Z 455.83,A -85,B 0,C 180,E1 -17521.621,E2 -17521.621} C_VEL
LIN {X 0,Y 292.243,Z 467.658,A -85,B 0,C 180,E1 -17522.618,E2 -17522.618} C_VEL
LIN {X 0,Y 290.17,Z 480.287,A -85,B 0,C 180,E1 -17523.971,E2 -17523.971} C_VEL
LIN {X 0,Y 287.917,Z 491.659,A -85,B 0,C 180,E1 -17525.483,E2 -17525.483} C_VEL
LIN {X 0,Y 285.619,Z 502.165,A -85,B 0,C 180,E1 -17527.198,E2 -17527.198} C_VEL
LIN {X 0,Y 283.235,Z 512.597,A -85,B 0,C 180,E1 -17529.293,E2 -17529.293} C_VEL
LIN {X 0,Y 281.129,Z 521.203,A -85,B 0,C 180,E1 -17531.414,E2 -17531.414} C_VEL
LIN {X 0,Y 279.367,Z 529.445,A -85,B 0,C 180,E1 -17533.935,E2 -17533.935} C_VEL
LIN {X 0,Y 277.904,Z 535.193,A -85,B 0,C 180,E1 -17536.099,E2 -17536.099} C_VEL
LIN {X 0,Y 276.878,Z 539.916,A -85,B 0,C 180,E1 -17538.284,E2 -17538.284} C_VEL
LIN {X 0,Y 275.935,Z 544.809,A -85,B 0,C 180,E1 -17541.21,E2 -17541.21} C_VEL
LIN {X 0,Y 275.451,Z 548.212,A -85,B 0,C 180,E1 -17544.142,E2 -17544.142} C_VEL
LIN {X 0,Y 275.269,Z 550.232,A -85,B 0,C 180,E1 -17547.073,E2 -17547.073} C_VEL
LIN {X 0,Y 275.22,Z 550.922,A -85,B 0,C 180,E1 -17550,E2 -17550} C_VEL
LIN {X 0,Y 275.269,Z 550.291,A -85,B 0,C 180,E1 -17552.927,E2 -17552.927} C_VEL
LIN {X 0,Y 275.491,Z 548.324,A -85,B 0,C 180,E1 -17555.857,E2 -17555.857} C_VEL
LIN {X 0,Y 275.932,Z 544.976,A -85,B 0,C 180,E1 -17558.79,E2 -17558.79} C_VEL
LIN {X 0,Y 276.852,Z 540.145,A -85,B 0,C 180,E1 -17561.717,E2 -17561.717} C_VEL
LIN {X 0,Y 277.87,Z 535.483,A -85,B 0,C 180,E1 -17563.903,E2 -17563.903} C_VEL
LIN {X 0,Y 279.477,Z 528.702,A -85,B 0,C 180,E1 -17566.433,E2 -17566.433} C_VEL
LIN {X 0,Y 281.381,Z 520.28,A -85,B 0,C 180,E1 -17568.947,E2 -17568.947} C_VEL
LIN {X 0,Y 283.543,Z 511.488,A -85,B 0,C 180,E1 -17571.063,E2 -17571.063} C_VEL
LIN {X 0,Y 285.949,Z 500.834,A -85,B 0,C 180,E1 -17573.156,E2 -17573.156} C_VEL
LIN {X 0,Y 288.339,Z 490.055,A -85,B 0,C 180,E1 -17574.862,E2 -17574.862} C_VEL
LIN {X 0,Y 290.468,Z 478.891,A -85,B 0,C 180,E1 -17576.311,E2 -17576.311} C_VEL
LIN {X 0,Y 292.369,Z 467.005,A -85,B 0,C 180,E1 -17577.563,E2 -17577.563} C_VEL
LIN {X 0,Y 294.181,Z 453.873,A -85,B 0,C 180,E1 -17578.638,E2 -17578.638} C_VEL
LIN {X 0,Y 295.78,Z 439.648,A -85,B 0,C 180,E1 -17579.491,E2 -17579.491} C_VEL
LIN {X 0,Y 296.829,Z 425.598,A -85,B 0,C 180,E1 -17580.06,E2 -17580.06} C_VEL
LIN {X 0,Y 299.036,Z 367.191,A -85,B 0,C 180,E1 -17581.446,E2 -17581.446} C_VEL
LIN {X 0,Y 300.021,Z 334.267,A -85,B 0,C 180,E1 -17582.24,E2 -17582.24} C_VEL
LIN {X 0,Y 293.583,Z 318.665,A -85,B 0,C 180,E1 -17583.485,E2 -17583.485} C_VEL
LIN {X 0,Y 285.263,Z 301.388,A -85,B 0,C 180,E1 -17585.119,E2 -17585.119} C_VEL
LIN {X 0,Y 278.877,Z 289.309,A -85,B 0,C 180,E1 -17586.468,E2 -17586.468} C_VEL
LIN {X 0,Y 277.289,Z 283.851,A -85,B 0,C 180,E1 -17588.592,E2 -17588.592} C_VEL
LIN {X 0,Y 277.228,Z 283.571,A -85,B 0,C 180,E1 -17589.328,E2 -17589.328} C_VEL
LIN {X 0,Y 277.214,Z 283.553,A -85,B 0,C 180,E1 -17593.196,E2 -17593.196} C_VEL
LIN {X 0,Y 277.216,Z 283.545,A -85,B 0,C 180,E1 -17597.324,E2 -17597.324} C_VEL
LIN {X 0,Y 277.275,Z 283.573,A -85,B 0,C 180,E1 -17601.788,E2 -17601.788} C_VEL
LIN {X 0,Y 277.3,Z 283.543,A -85,B 0,C 180,E1 -17604.343,E2 -17604.343} C_VEL
LIN {X 0,Y 277.24,Z 283.527,A -85,B 0,C 180,E1 -17607.836,E2 -17607.836} C_VEL
LIN {X 0,Y 277.228,Z 283.545,A -85,B 0,C 180,E1 -17608.829,E2 -17608.829} C_VEL
LIN {X 0,Y 276.584,Z 283.651,A -85,B 0,C 180,E1 -17610.041,E2 -17610.041} C_VEL
LIN {X 0,Y 273.726,Z 284.014,A -85,B 0,C 180,E1 -17612.017,E2 -17612.017} C_VEL
LIN {X 0,Y 271.312,Z 284.304,A -85,B 0,C 180,E1 -17613.622,E2 -17613.622} C_VEL
LIN {X 0,Y 270.318,Z 284.426,A -85,B 0,C 180,E1 -17614.867,E2 -17614.867} C_VEL
LIN {X 0,Y 270.261,Z 284.438,A -85,B 0,C 180,E1 -17615.288,E2 -17615.288} C_VEL
LIN {X 0,Y 270.297,Z 284.427,A -85,B 0,C 180,E1 -17620.244,E2 -17620.244} C_VEL
LIN {X 0,Y 270.391,Z 284.408,A -85,B 0,C 180,E1 -17624.935,E2 -17624.935} C_VEL
LIN {X 0,Y 270.407,Z 284.419,A -85,B 0,C 180,E1 -17629.517,E2 -17629.517} C_VEL
LIN {X 0,Y 270.593,Z 284.39,A -85,B 0,C 180,E1 -17632.538,E2 -17632.538} C_VEL
LIN {X 0,Y 270.782,Z 284.359,A -85,B 0,C 180,E1 -17638.513,E2 -17638.513} C_VEL
LIN {X 0,Y 270.782,Z 284.378,A -85,B 0,C 180,E1 -17641.487,E2 -17641.487} C_VEL
LIN {X 0,Y 270.605,Z 284.401,A -85,B 0,C 180,E1 -17647.461,E2 -17647.461} C_VEL
LIN {X 0,Y 270.436,Z 284.402,A -85,B 0,C 180,E1 -17650.481,E2 -17650.481} C_VEL
LIN {X 0,Y 270.391,Z 284.419,A -85,B 0,C 180,E1 -17655.065,E2 -17655.065} C_VEL
LIN {X 0,Y 270.296,Z 284.442,A -85,B 0,C 180,E1 -17659.756,E2 -17659.756} C_VEL
LIN {X 0,Y 270.269,Z 284.445,A -85,B 0,C 180,E1 -17664.586,E2 -17664.586} C_VEL
LIN {X 0,Y 270.267,Z 284.429,A -85,B 0,C 180,E1 -17667.909,E2 -17667.909} C_VEL
LIN {X 0,Y 270.18,Z 284.442,A -85,B 0,C 180,E1 -17671.349,E2 -17671.349} C_VEL
LIN {X 0,Y 270.198,Z 284.397,A -85,B 0,C 180,E1 -17674.906,E2 -17674.906} C_VEL
LIN {X 0,Y 270.194,Z 284.454,A -85,B 0,C 180,E1 -17678.711,E2 -17678.711} C_VEL
LIN {X 0,Y 270.186,Z 284.449,A -85,B 0,C 180,E1 -17683.255,E2 -17683.255} C_VEL
LIN {X 0,Y 270.22,Z 284.424,A -85,B 0,C 180,E1 -17687.452,E2 -17687.452} C_VEL
LIN {X 0,Y 270.268,Z 284.557,A -85,B 0,C 180,E1 -17689.087,E2 -17689.087} C_VEL
LIN {X 0,Y 272.572,Z 292.92,A -85,B 0,C 180,E1 -17692.515,E2 -17692.515} C_VEL
LIN {X 0,Y 274.016,Z 296.138,A -85,B 0,C 180,E1 -17692.952,E2 -17692.952} C_VEL
LIN {X 0,Y 279.9,Z 307.189,A -85,B 0,C 180,E1 -17694.197,E2 -17694.197} C_VEL
LIN {X 0,Y 288.039,Z 324.583,A -85,B 0,C 180,E1 -17695.869,E2 -17695.869} C_VEL
LIN {X 0,Y 292.583,Z 335.676,A -85,B 0,C 180,E1 -17696.789,E2 -17696.789} C_VEL
LIN {X 0,Y 293.869,Z 343.891,A -85,B 0,C 180,E1 -17697.187,E2 -17697.187} C_VEL
LIN {X 0,Y 290.62,Z 430.52,A -85,B 0,C 180,E1 -17699.282,E2 -17699.282} C_VEL
LIN {X 0,Y 289.349,Z 445.241,A -85,B 0,C 180,E1 -17699.887,E2 -17699.887} C_VEL
LIN {X 0,Y 287.676,Z 459.263,A -85,B 0,C 180,E1 -17700.752,E2 -17700.752} C_VEL
LIN {X 0,Y 285.555,Z 473.159,A -85,B 0,C 180,E1 -17701.921,E2 -17701.921} C_VEL
LIN {X 0,Y 283.277,Z 485.87,A -85,B 0,C 180,E1 -17703.316,E2 -17703.316} C_VEL
LIN {X 0,Y 280.814,Z 498.141,A -85,B 0,C 180,E1 -17705.019,E2 -17705.019} C_VEL
LIN {X 0,Y 278.172,Z 509.311,A -85,B 0,C 180,E1 -17706.946,E2 -17706.946} C_VEL
LIN {X 0,Y 275.74,Z 519.335,A -85,B 0,C 180,E1 -17709.095,E2 -17709.095} C_VEL
LIN {X 0,Y 273.691,Z 527.66,A -85,B 0,C 180,E1 -17711.278,E2 -17711.278} C_VEL
LIN {X 0,Y 271.789,Z 535.62,A -85,B 0,C 180,E1 -17713.861,E2 -17713.861} C_VEL
LIN {X 0,Y 270.267,Z 542.029,A -85,B 0,C 180,E1 -17716.466,E2 -17716.466} C_VEL
LIN {X 0,Y 269.077,Z 547.711,A -85,B 0,C 180,E1 -17719.466,E2 -17719.466} C_VEL
LIN {X 0,Y 268.425,Z 551.833,A -85,B 0,C 180,E1 -17722.478,E2 -17722.478} C_VEL
LIN {X 0,Y 268.131,Z 554.524,A -85,B 0,C 180,E1 -17725.49,E2 -17725.49} C_VEL
LIN {X 0,Y 268.126,Z 555.855,A -85,B 0,C 180,E1 -17728.498,E2 -17728.498} C_VEL
LIN {X 0,Y 268.126,Z 555.848,A -85,B 0,C 180,E1 -17731.502,E2 -17731.502} C_VEL
LIN {X 0,Y 268.131,Z 554.505,A -85,B 0,C 180,E1 -17734.51,E2 -17734.51} C_VEL
LIN {X 0,Y 268.425,Z 551.802,A -85,B 0,C 180,E1 -17737.522,E2 -17737.522} C_VEL
LIN {X 0,Y 269.095,Z 547.662,A -85,B 0,C 180,E1 -17740.534,E2 -17740.534} C_VEL
LIN {X 0,Y 270.267,Z 541.962,A -85,B 0,C 180,E1 -17743.535,E2 -17743.535} C_VEL
LIN {X 0,Y 271.762,Z 535.539,A -85,B 0,C 180,E1 -17746.141,E2 -17746.141} C_VEL
LIN {X 0,Y 273.621,Z 527.558,A -85,B 0,C 180,E1 -17748.727,E2 -17748.727} C_VEL
LIN {X 0,Y 275.727,Z 519.211,A -85,B 0,C 180,E1 -17750.906,E2 -17750.906} C_VEL
LIN {X 0,Y 278.117,Z 509.162,A -85,B 0,C 180,E1 -17753.059,E2 -17753.059} C_VEL
LIN {X 0,Y 280.831,Z 497.946,A -85,B 0,C 180,E1 -17754.98,E2 -17754.98} C_VEL
LIN {X 0,Y 283.082,Z 486.786,A -85,B 0,C 180,E1 -17756.543,E2 -17756.543} C_VEL
LIN {X 0,Y 285.278,Z 474.626,A -85,B 0,C 180,E1 -17757.909,E2 -17757.909} C_VEL
LIN {X 0,Y 287.369,Z 461.125,A -85,B 0,C 180,E1 -17759.082,E2 -17759.082} C_VEL
LIN {X 0,Y 289.144,Z 446.992,A -85,B 0,C 180,E1 -17759.986,E2 -17759.986} C_VEL
LIN {X 0,Y 290.311,Z 433.162,A -85,B 0,C 180,E1 -17760.604,E2 -17760.604} C_VEL
LIN {X 0,Y 291.365,Z 411.597,A -85,B 0,C 180,E1 -17761.166,E2 -17761.166} C_VEL
LIN {X 0,Y 293.716,Z 343.411,A -85,B 0,C 180,E1 -17762.811,E2 -17762.811} C_VEL
LIN {X 0,Y 292.254,Z 334.673,A -85,B 0,C 180,E1 -17763.246,E2 -17763.246} C_VEL
LIN {X 0,Y 285.062,Z 317.958,A -85,B 0,C 180,E1 -17764.695,E2 -17764.695} C_VEL
LIN {X 0,Y 276.947,Z 301.454,A -85,B 0,C 180,E1 -17766.381,E2 -17766.381} C_VEL
LIN {X 0,Y 272.663,Z 293.282,A -85,B 0,C 180,E1 -17767.354,E2 -17767.354} C_VEL
LIN {X 0,Y 270.326,Z 285.191,A -85,B 0,C 180,E1 -17770.537,E2 -17770.537} C_VEL
LIN {X 0,Y 270.19,Z 284.451,A -85,B 0,C 180,E1 -17771.033,E2 -17771.033} C_VEL
LIN {X 0,Y 270.149,Z 284.452,A -85,B 0,C 180,E1 -17775.379,E2 -17775.379} C_VEL
LIN {X 0,Y 270.171,Z 284.445,A -85,B 0,C 180,E1 -17779.434,E2 -17779.434} C_VEL
LIN {X 0,Y 270.223,Z 284.408,A -85,B 0,C 180,E1 -17783.73,E2 -17783.73} C_VEL
LIN {X 0,Y 270.199,Z 284.405,A -85,B 0,C 180,E1 -17786.892,E2 -17786.892} C_VEL
LIN {X 0,Y 270.225,Z 284.449,A -85,B 0,C 180,E1 -17790.386,E2 -17790.386} C_VEL
LIN {X 0,Y 270.26,Z 284.436,A -85,B 0,C 180,E1 -17793.764,E2 -17793.764} C_VEL
LIN {X 0,Y 270.228,Z 284.434,A -85,B 0,C 180,E1 -17797.038,E2 -17797.038} C_VEL
LIN {X 0,Y 270.297,Z 284.442,A -85,B 0,C 180,E1 -17800.244,E2 -17800.244} C_VEL
LIN {X 0,Y 270.391,Z 284.419,A -85,B 0,C 180,E1 -17804.935,E2 -17804.935} C_VEL
LIN {X 0,Y 270.437,Z 284.401,A -85,B 0,C 180,E1 -17809.519,E2 -17809.519} C_VEL
LIN {X 0,Y 270.606,Z 284.401,A -85,B 0,C 180,E1 -17812.539,E2 -17812.539} C_VEL
LIN {X 0,Y 270.782,Z 284.378,A -85,B 0,C 180,E1 -17818.513,E2 -17818.513} C_VEL
LIN {X 0,Y 270.782,Z 284.36,A -85,B 0,C 180,E1 -17821.487,E2 -17821.487} C_VEL
LIN {X 0,Y 270.594,Z 284.39,A -85,B 0,C 180,E1 -17827.462,E2 -17827.462} C_VEL
LIN {X 0,Y 270.408,Z 284.417,A -85,B 0,C 180,E1 -17830.482,E2 -17830.482} C_VEL
LIN {X 0,Y 270.392,Z 284.408,A -85,B 0,C 180,E1 -17835.065,E2 -17835.065} C_VEL
LIN {X 0,Y 270.297,Z 284.428,A -85,B 0,C 180,E1 -17839.756,E2 -17839.756} C_VEL
LIN {X 0,Y 270.27,Z 284.44,A -85,B 0,C 180,E1 -17844.586,E2 -17844.586} C_VEL
LIN {X 0,Y 270.269,Z 284.44,A -85,B 0,C 180,E1 -17847.909,E2 -17847.909} C_VEL
LIN {X 0,Y 270.181,Z 284.418,A -85,B 0,C 180,E1 -17851.349,E2 -17851.349} C_VEL
LIN {X 0,Y 270.212,Z 284.402,A -85,B 0,C 180,E1 -17854.904,E2 -17854.904} C_VEL
LIN {X 0,Y 270.22,Z 284.443,A -85,B 0,C 180,E1 -17858.718,E2 -17858.718} C_VEL
LIN {X 0,Y 270.17,Z 284.427,A -85,B 0,C 180,E1 -17863.251,E2 -17863.251} C_VEL
LIN {X 0,Y 270.173,Z 284.427,A -85,B 0,C 180,E1 -17867.443,E2 -17867.443} C_VEL
LIN {X 0,Y 270.208,Z 284.573,A -85,B 0,C 180,E1 -17870.537,E2 -17870.537} C_VEL
LIN {X 0,Y 271.559,Z 289.283,A -85,B 0,C 180,E1 -17872.503,E2 -17872.503} C_VEL
LIN {X 0,Y 276.695,Z 298.779,A -85,B 0,C 180,E1 -17873.673,E2 -17873.673} C_VEL
LIN {X 0,Y 283.977,Z 313.028,A -85,B 0,C 180,E1 -17875.182,E2 -17875.182} C_VEL
LIN {X 0,Y 291.979,Z 330.989,A -85,B 0,C 180,E1 -17876.789,E2 -17876.789} C_VEL
LIN {X 0,Y 293.963,Z 336.152,A -85,B 0,C 180,E1 -17877.19,E2 -17877.19} C_VEL
LIN {X 0,Y 291.285,Z 411.676,A -85,B 0,C 180,E1 -17879.004,E2 -17879.004} C_VEL
LIN {X 0,Y 290.439,Z 429.699,A -85,B 0,C 180,E1 -17879.51,E2 -17879.51} C_VEL
LIN {X 0,Y 289.197,Z 443.133,A -85,B 0,C 180,E1 -17880.121,E2 -17880.121} C_VEL
LIN {X 0,Y 287.508,Z 457.033,A -85,B 0,C 180,E1 -17881.033,E2 -17881.033} C_VEL
LIN {X 0,Y 285.662,Z 469.496,A -85,B 0,C 180,E1 -17882.132,E2 -17882.132} C_VEL
LIN {X 0,Y 283.56,Z 481.709,A -85,B 0,C 180,E1 -17883.505,E2 -17883.505} C_VEL
LIN {X 0,Y 281.229,Z 492.901,A -85,B 0,C 180,E1 -17885.058,E2 -17885.058} C_VEL
LIN {X 0,Y 278.628,Z 504.153,A -85,B 0,C 180,E1 -17886.986,E2 -17886.986} C_VEL
LIN {X 0,Y 276.187,Z 514.205,A -85,B 0,C 180,E1 -17889.13,E2 -17889.13} C_VEL
LIN {X 0,Y 274.05,Z 522.554,A -85,B 0,C 180,E1 -17891.304,E2 -17891.304} C_VEL
LIN {X 0,Y 272.286,Z 530.52,A -85,B 0,C 180,E1 -17893.891,E2 -17893.891} C_VEL
LIN {X 0,Y 270.529,Z 536.937,A -85,B 0,C 180,E1 -17896.479,E2 -17896.479} C_VEL
LIN {X 0,Y 269.324,Z 542.625,A -85,B 0,C 180,E1 -17899.475,E2 -17899.475} C_VEL
LIN {X 0,Y 268.62,Z 546.756,A -85,B 0,C 180,E1 -17902.483,E2 -17902.483} C_VEL
LIN {X 0,Y 268.223,Z 549.458,A -85,B 0,C 180,E1 -17905.492,E2 -17905.492} C_VEL
LIN {X 0,Y 268.143,Z 550.809,A -85,B 0,C 180,E1 -17908.498,E2 -17908.498} C_VEL
LIN {X 0,Y 268.143,Z 550.838,A -85,B 0,C 180,E1 -17911.502,E2 -17911.502} C_VEL
LIN {X 0,Y 268.227,Z 549.544,A -85,B 0,C 180,E1 -17914.508,E2 -17914.508} C_VEL
LIN {X 0,Y 268.603,Z 546.894,A -85,B 0,C 180,E1 -17917.517,E2 -17917.517} C_VEL
LIN {X 0,Y 269.295,Z 542.821,A -85,B 0,C 180,E1 -17920.526,E2 -17920.526} C_VEL
LIN {X 0,Y 270.501,Z 537.194,A -85,B 0,C 180,E1 -17923.522,E2 -17923.522} C_VEL
LIN {X 0,Y 272.191,Z 530.838,A -85,B 0,C 180,E1 -17926.115,E2 -17926.115} C_VEL
LIN {X 0,Y 273.947,Z 523.184,A -85,B 0,C 180,E1 -17928.626,E2 -17928.626} C_VEL
LIN {X 0,Y 276.086,Z 514.671,A -85,B 0,C 180,E1 -17930.878,E2 -17930.878} C_VEL
LIN {X 0,Y 278.566,Z 504.71,A -85,B 0,C 180,E1 -17933.019,E2 -17933.019} C_VEL
LIN {X 0,Y 281.139,Z 493.62,A -85,B 0,C 180,E1 -17934.95,E2 -17934.95} C_VEL
LIN {X 0,Y 283.491,Z 482.576,A -85,B 0,C 180,E1 -17936.502,E2 -17936.502} C_VEL
LIN {X 0,Y 285.539,Z 470.584,A -85,B 0,C 180,E1 -17937.881,E2 -17937.881} C_VEL
LIN {X 0,Y 287.566,Z 457.318,A -85,B 0,C 180,E1 -17939.06,E2 -17939.06} C_VEL
LIN {X 0,Y 289.212,Z 443.514,A -85,B 0,C 180,E1 -17939.978,E2 -17939.978} C_VEL
LIN {X 0,Y 290.495,Z 429.145,A -85,B 0,C 180,E1 -17940.633,E2 -17940.633} C_VEL
LIN {X 0,Y 291.48,Z 409.371,A -85,B 0,C 180,E1 -17941.163,E2 -17941.163} C_VEL
LIN {X 0,Y 293.99,Z 336.111,A -85,B 0,C 180,E1 -17942.933,E2 -17942.933} C_VEL
LIN {X 0,Y 287.57,Z 320.773,A -85,B 0,C 180,E1 -17944.22,E2 -17944.22} C_VEL
LIN {X 0,Y 280.24,Z 305.471,A -85,B 0,C 180,E1 -17945.719,E2 -17945.719} C_VEL
LIN {X 0,Y 273.243,Z 292.555,A -85,B 0,C 180,E1 -17947.199,E2 -17947.199} C_VEL
LIN {X 0,Y 271.515,Z 289.093,A -85,B 0,C 180,E1 -17947.675,E2 -17947.675} C_VEL
LIN {X 0,Y 270.194,Z 284.527,A -85,B 0,C 180,E1 -17949.647,E2 -17949.647} C_VEL
LIN {X 0,Y 270.169,Z 284.431,A -85,B 0,C 180,E1 -17953.25,E2 -17953.25} C_VEL
LIN {X 0,Y 270.172,Z 284.42,A -85,B 0,C 180,E1 -17957.441,E2 -17957.441} C_VEL
LIN {X 0,Y 270.204,Z 284.448,A -85,B 0,C 180,E1 -17961.373,E2 -17961.373} C_VEL
LIN {X 0,Y 270.211,Z 284.408,A -85,B 0,C 180,E1 -17965.096,E2 -17965.096} C_VEL
LIN {X 0,Y 270.196,Z 284.427,A -85,B 0,C 180,E1 -17969.13,E2 -17969.13} C_VEL
LIN {X 0,Y 270.261,Z 284.445,A -85,B 0,C 180,E1 -17972.145,E2 -17972.145} C_VEL
LIN {X 0,Y 270.261,Z 284.438,A -85,B 0,C 180,E1 -17975.288,E2 -17975.288} C_VEL
LIN {X 0,Y 269.653,Z 284.526,A -85,B 0,C 180,E1 -17976.533,E2 -17976.533} C_VEL
LIN {X 0,Y 266.812,Z 284.883,A -85,B 0,C 180,E1 -17978.561,E2 -17978.561} C_VEL
LIN {X 0,Y 264.364,Z 285.181,A -85,B 0,C 180,E1 -17980.21,E2 -17980.21} C_VEL
LIN {X 0,Y 263.312,Z 285.311,A -85,B 0,C 180,E1 -17981.489,E2 -17981.489} C_VEL
LIN {X 0,Y 263.228,Z 285.315,A -85,B 0,C 180,E1 -17981.923,E2 -17981.923} C_VEL
LIN {X 0,Y 263.339,Z 285.287,A -85,B 0,C 180,E1 -17984.521,E2 -17984.521} C_VEL
LIN {X 0,Y 263.349,Z 285.3,A -85,B 0,C 180,E1 -17989.233,E2 -17989.233} C_VEL
LIN {X 0,Y 263.553,Z 285.264,A -85,B 0,C 180,E1 -17992.338,E2 -17992.338} C_VEL
LIN {X 0,Y 263.746,Z 285.235,A -85,B 0,C 180,E1 -17998.473,E2 -17998.473} C_VEL
LIN {X 0,Y 263.746,Z 285.255,A -85,B 0,C 180,E1 -18001.527,E2 -18001.527} C_VEL
LIN {X 0,Y 263.566,Z 285.278,A -85,B 0,C 180,E1 -18007.662,E2 -18007.662} C_VEL
LIN {X 0,Y 263.368,Z 285.282,A -85,B 0,C 180,E1 -18010.766,E2 -18010.766} C_VEL
LIN {X 0,Y 263.339,Z 285.292,A -85,B 0,C 180,E1 -18015.479,E2 -18015.479} C_VEL
LIN {X 0,Y 263.258,Z 285.312,A -85,B 0,C 180,E1 -18020.307,E2 -18020.307} C_VEL
LIN {X 0,Y 263.204,Z 285.324,A -85,B 0,C 180,E1 -18025.292,E2 -18025.292} C_VEL
LIN {X 0,Y 263.175,Z 285.32,A -85,B 0,C 180,E1 -18028.73,E2 -18028.73} C_VEL
LIN {X 0,Y 263.128,Z 285.297,A -85,B 0,C 180,E1 -18032.289,E2 -18032.289} C_VEL
LIN {X 0,Y 263.181,Z 285.296,A -85,B 0,C 180,E1 -18036.764,E2 -18036.764} C_VEL
LIN {X 0,Y 263.128,Z 285.328,A -85,B 0,C 180,E1 -18041.596,E2 -18041.596} C_VEL
LIN {X 0,Y 263.142,Z 285.328,A -85,B 0,C 180,E1 -18046.021,E2 -18046.021} C_VEL
LIN {X 0,Y 263.2,Z 285.533,A -85,B 0,C 180,E1 -18048.185,E2 -18048.185} C_VEL
LIN {X 0,Y 265.29,Z 292.924,A -85,B 0,C 180,E1 -18051.322,E2 -18051.322} C_VEL
LIN {X 0,Y 267.556,Z 297.187,A -85,B 0,C 180,E1 -18051.937,E2 -18051.937} C_VEL
LIN {X 0,Y 275.592,Z 312.665,A -85,B 0,C 180,E1 -18053.723,E2 -18053.723} C_VEL
LIN {X 0,Y 283.721,Z 330.337,A -85,B 0,C 180,E1 -18055.451,E2 -18055.451} C_VEL
LIN {X 0,Y 286.876,Z 338.32,A -85,B 0,C 180,E1 -18056.119,E2 -18056.119} C_VEL
LIN {X 0,Y 287.884,Z 345.098,A -85,B 0,C 180,E1 -18056.452,E2 -18056.452} C_VEL
LIN {X 0,Y 284.533,Z 430.644,A -85,B 0,C 180,E1 -18058.558,E2 -18058.558} C_VEL
LIN {X 0,Y 283.236,Z 445.184,A -85,B 0,C 180,E1 -18059.167,E2 -18059.167} C_VEL
LIN {X 0,Y 281.521,Z 459.203,A -85,B 0,C 180,E1 -18060.048,E2 -18060.048} C_VEL
LIN {X 0,Y 279.607,Z 471.331,A -85,B 0,C 180,E1 -18061.063,E2 -18061.063} C_VEL
LIN {X 0,Y 277.286,Z 484.115,A -85,B 0,C 180,E1 -18062.449,E2 -18062.449} C_VEL
LIN {X 0,Y 274.861,Z 495.821,A -85,B 0,C 180,E1 -18064.048,E2 -18064.048} C_VEL
LIN {X 0,Y 272.089,Z 507.357,A -85,B 0,C 180,E1 -18065.995,E2 -18065.995} C_VEL
LIN {X 0,Y 269.489,Z 517.755,A -85,B 0,C 180,E1 -18068.185,E2 -18068.185} C_VEL
LIN {X 0,Y 267.235,Z 526.333,A -85,B 0,C 180,E1 -18070.409,E2 -18070.409} C_VEL
LIN {X 0,Y 265.241,Z 534.546,A -85,B 0,C 180,E1 -18073.055,E2 -18073.055} C_VEL
LIN {X 0,Y 263.783,Z 540.299,A -85,B 0,C 180,E1 -18075.339,E2 -18075.339} C_VEL
LIN {X 0,Y 262.56,Z 545.008,A -85,B 0,C 180,E1 -18077.635,E2 -18077.635} C_VEL
LIN {X 0,Y 261.683,Z 549.891,A -85,B 0,C 180,E1 -18080.727,E2 -18080.727} C_VEL
LIN {X 0,Y 261.152,Z 553.285,A -85,B 0,C 180,E1 -18083.821,E2 -18083.821} C_VEL
LIN {X 0,Y 261.006,Z 555.292,A -85,B 0,C 180,E1 -18086.913,E2 -18086.913} C_VEL
LIN {X 0,Y 261.072,Z 555.952,A -85,B 0,C 180,E1 -18090,E2 -18090} C_VEL
LIN {X 0,Y 261.007,Z 555.277,A -85,B 0,C 180,E1 -18093.087,E2 -18093.087} C_VEL
LIN {X 0,Y 261.163,Z 553.26,A -85,B 0,C 180,E1 -18096.179,E2 -18096.179} C_VEL
LIN {X 0,Y 261.683,Z 549.851,A -85,B 0,C 180,E1 -18099.273,E2 -18099.273} C_VEL
LIN {X 0,Y 262.562,Z 544.947,A -85,B 0,C 180,E1 -18102.365,E2 -18102.365} C_VEL
LIN {X 0,Y 264.244,Z 538.409,A -85,B 0,C 180,E1 -18105.424,E2 -18105.424} C_VEL
LIN {X 0,Y 265.796,Z 531.554,A -85,B 0,C 180,E1 -18107.95,E2 -18107.95} C_VEL
LIN {X 0,Y 267.911,Z 523.505,A -85,B 0,C 180,E1 -18110.339,E2 -18110.339} C_VEL
LIN {X 0,Y 270.303,Z 514.357,A -85,B 0,C 180,E1 -18112.551,E2 -18112.551} C_VEL
LIN {X 0,Y 272.57,Z 505.235,A -85,B 0,C 180,E1 -18114.364,E2 -18114.364} C_VEL
LIN {X 0,Y 275.396,Z 493.478,A -85,B 0,C 180,E1 -18116.269,E2 -18116.269} C_VEL
LIN {X 0,Y 277.524,Z 482.582,A -85,B 0,C 180,E1 -18117.71,E2 -18117.71} C_VEL
LIN {X 0,Y 279.935,Z 469.234,A -85,B 0,C 180,E1 -18119.105,E2 -18119.105} C_VEL
LIN {X 0,Y 282.03,Z 455.207,A -85,B 0,C 180,E1 -18120.202,E2 -18120.202} C_VEL
LIN {X 0,Y 283.577,Z 441.16,A -85,B 0,C 180,E1 -18120.999,E2 -18120.999} C_VEL
LIN {X 0,Y 284.702,Z 426.973,A -85,B 0,C 180,E1 -18121.514,E2 -18121.514} C_VEL
LIN {X 0,Y 287.796,Z 344.752,A -85,B 0,C 180,E1 -18123.532,E2 -18123.532} C_VEL
LIN {X 0,Y 286.568,Z 337.363,A -85,B 0,C 180,E1 -18123.912,E2 -18123.912} C_VEL
LIN {X 0,Y 278.904,Z 319.512,A -85,B 0,C 180,E1 -18125.525,E2 -18125.525} C_VEL
LIN {X 0,Y 269.929,Z 301.602,A -85,B 0,C 180,E1 -18127.478,E2 -18127.478} C_VEL
LIN {X 0,Y 265.342,Z 293.143,A -85,B 0,C 180,E1 -18128.579,E2 -18128.579} C_VEL
LIN {X 0,Y 263.195,Z 285.818,A -85,B 0,C 180,E1 -18131.611,E2 -18131.611} C_VEL
LIN {X 0,Y 263.123,Z 285.305,A -85,B 0,C 180,E1 -18132.15,E2 -18132.15} C_VEL
LIN {X 0,Y 263.102,Z 285.328,A -85,B 0,C 180,E1 -18136.155,E2 -18136.155} C_VEL
LIN {X 0,Y 263.102,Z 285.328,A -85,B 0,C 180,E1 -18140.127,E2 -18140.127} C_VEL
LIN {X 0,Y 263.16,Z 285.282,A -85,B 0,C 180,E1 -18144.018,E2 -18144.018} C_VEL
LIN {X 0,Y 263.129,Z 285.299,A -85,B 0,C 180,E1 -18147.711,E2 -18147.711} C_VEL
LIN {X 0,Y 263.197,Z 285.311,A -85,B 0,C 180,E1 -18151.783,E2 -18151.783} C_VEL
LIN {X 0,Y 263.222,Z 285.322,A -85,B 0,C 180,E1 -18155.2,E2 -18155.2} C_VEL
LIN {X 0,Y 263.259,Z 285.313,A -85,B 0,C 180,E1 -18159.693,E2 -18159.693} C_VEL
LIN {X 0,Y 263.34,Z 285.292,A -85,B 0,C 180,E1 -18164.521,E2 -18164.521} C_VEL
LIN {X 0,Y 263.369,Z 285.282,A -85,B 0,C 180,E1 -18169.234,E2 -18169.234} C_VEL
LIN {X 0,Y 263.567,Z 285.278,A -85,B 0,C 180,E1 -18172.338,E2 -18172.338} C_VEL
LIN {X 0,Y 263.746,Z 285.255,A -85,B 0,C 180,E1 -18178.473,E2 -18178.473} C_VEL
LIN {X 0,Y 263.746,Z 285.235,A -85,B 0,C 180,E1 -18181.527,E2 -18181.527} C_VEL
LIN {X 0,Y 263.553,Z 285.265,A -85,B 0,C 180,E1 -18187.662,E2 -18187.662} C_VEL
LIN {X 0,Y 263.35,Z 285.299,A -85,B 0,C 180,E1 -18190.767,E2 -18190.767} C_VEL
LIN {X 0,Y 263.34,Z 285.287,A -85,B 0,C 180,E1 -18195.479,E2 -18195.479} C_VEL
LIN {X 0,Y 263.26,Z 285.3,A -85,B 0,C 180,E1 -18200.307,E2 -18200.307} C_VEL
LIN {X 0,Y 263.205,Z 285.311,A -85,B 0,C 180,E1 -18205.292,E2 -18205.292} C_VEL
LIN {X 0,Y 263.177,Z 285.329,A -85,B 0,C 180,E1 -18208.73,E2 -18208.73} C_VEL
LIN {X 0,Y 263.13,Z 285.279,A -85,B 0,C 180,E1 -18212.289,E2 -18212.289} C_VEL
LIN {X 0,Y 263.185,Z 285.297,A -85,B 0,C 180,E1 -18215.979,E2 -18215.979} C_VEL
LIN {X 0,Y 263.113,Z 285.303,A -85,B 0,C 180,E1 -18219.871,E2 -18219.871} C_VEL
LIN {X 0,Y 263.126,Z 285.318,A -85,B 0,C 180,E1 -18223.984,E2 -18223.984} C_VEL
LIN {X 0,Y 263.123,Z 285.307,A -85,B 0,C 180,E1 -18228.407,E2 -18228.407} C_VEL
LIN {X 0,Y 263.155,Z 285.521,A -85,B 0,C 180,E1 -18229.637,E2 -18229.637} C_VEL
LIN {X 0,Y 264.286,Z 289.372,A -85,B 0,C 180,E1 -18231.281,E2 -18231.281} C_VEL
LIN {X 0,Y 271.467,Z 302.236,A -85,B 0,C 180,E1 -18232.968,E2 -18232.968} C_VEL
LIN {X 0,Y 280.439,Z 320.263,A -85,B 0,C 180,E1 -18234.898,E2 -18234.898} C_VEL
LIN {X 0,Y 287.194,Z 335.992,A -85,B 0,C 180,E1 -18236.308,E2 -18236.308} C_VEL
LIN {X 0,Y 287.944,Z 338.038,A -85,B 0,C 180,E1 -18236.467,E2 -18236.467} C_VEL
LIN {X 0,Y 285.383,Z 407.772,A -85,B 0,C 180,E1 -18238.173,E2 -18238.173} C_VEL
LIN {X 0,Y 284.428,Z 428.642,A -85,B 0,C 180,E1 -18238.743,E2 -18238.743} C_VEL
LIN {X 0,Y 283.06,Z 443.209,A -85,B 0,C 180,E1 -18239.404,E2 -18239.404} C_VEL
LIN {X 0,Y 281.317,Z 457.107,A -85,B 0,C 180,E1 -18240.333,E2 -18240.333} C_VEL
LIN {X 0,Y 279.41,Z 469.568,A -85,B 0,C 180,E1 -18241.452,E2 -18241.452} C_VEL
LIN {X 0,Y 277.217,Z 481.781,A -85,B 0,C 180,E1 -18242.85,E2 -18242.85} C_VEL
LIN {X 0,Y 274.791,Z 492.972,A -85,B 0,C 180,E1 -18244.432,E2 -18244.432} C_VEL
LIN {X 0,Y 272.089,Z 504.223,A -85,B 0,C 180,E1 -18246.4,E2 -18246.4} C_VEL
LIN {X 0,Y 269.536,Z 514.275,A -85,B 0,C 180,E1 -18248.59,E2 -18248.59} C_VEL
LIN {X 0,Y 267.314,Z 522.62,A -85,B 0,C 180,E1 -18250.814,E2 -18250.814} C_VEL
LIN {X 0,Y 265.43,Z 530.589,A -85,B 0,C 180,E1 -18253.463,E2 -18253.463} C_VEL
LIN {X 0,Y 263.608,Z 537.005,A -85,B 0,C 180,E1 -18256.117,E2 -18256.117} C_VEL
LIN {X 0,Y 262.33,Z 542.692,A -85,B 0,C 180,E1 -18259.191,E2 -18259.191} C_VEL
LIN {X 0,Y 261.559,Z 546.824,A -85,B 0,C 180,E1 -18262.279,E2 -18262.279} C_VEL
LIN {X 0,Y 261.144,Z 549.525,A -85,B 0,C 180,E1 -18265.369,E2 -18265.369} C_VEL
LIN {X 0,Y 261.052,Z 550.875,A -85,B 0,C 180,E1 -18268.457,E2 -18268.457} C_VEL
LIN {X 0,Y 261.075,Z 551.055,A -85,B 0,C 180,E1 -18270,E2 -18270} C_VEL
LIN {X 0,Y 261.082,Z 550.424,A -85,B 0,C 180,E1 -18273.086,E2 -18273.086} C_VEL
LIN {X 0,Y 261.321,Z 548.457,A -85,B 0,C 180,E1 -18276.175,E2 -18276.175} C_VEL
LIN {X 0,Y 261.863,Z 545.108,A -85,B 0,C 180,E1 -18279.266,E2 -18279.266} C_VEL
LIN {X 0,Y 262.901,Z 540.277,A -85,B 0,C 180,E1 -18282.348,E2 -18282.348} C_VEL
LIN {X 0,Y 264.069,Z 535.613,A -85,B 0,C 180,E1 -18284.645,E2 -18284.645} C_VEL
LIN {X 0,Y 265.525,Z 529.899,A -85,B 0,C 180,E1 -18286.926,E2 -18286.926} C_VEL
LIN {X 0,Y 267.608,Z 521.758,A -85,B 0,C 180,E1 -18289.563,E2 -18289.563} C_VEL
LIN {X 0,Y 269.883,Z 513.237,A -85,B 0,C 180,E1 -18291.782,E2 -18291.782} C_VEL
LIN {X 0,Y 272.46,Z 502.909,A -85,B 0,C 180,E1 -18293.97,E2 -18293.97} C_VEL
LIN {X 0,Y 275.25,Z 491.353,A -85,B 0,C 180,E1 -18295.928,E2 -18295.928} C_VEL
LIN {X 0,Y 277.632,Z 479.734,A -85,B 0,C 180,E1 -18297.525,E2 -18297.525} C_VEL
LIN {X 0,Y 279.853,Z 467.126,A -85,B 0,C 180,E1 -18298.909,E2 -18298.909} C_VEL
LIN {X 0,Y 281.83,Z 453.991,A -85,B 0,C 180,E1 -18300.019,E2 -18300.019} C_VEL
LIN {X 0,Y 283.508,Z 439.761,A -85,B 0,C 180,E1 -18300.903,E2 -18300.903} C_VEL
LIN {X 0,Y 284.617,Z 426.008,A -85,B 0,C 180,E1 -18301.48,E2 -18301.48} C_VEL
LIN {X 0,Y 287.042,Z 367.047,A -85,B 0,C 180,E1 -18302.929,E2 -18302.929} C_VEL
LIN {X 0,Y 288.055,Z 338.416,A -85,B 0,C 180,E1 -18303.635,E2 -18303.635} C_VEL
LIN {X 0,Y 282.801,Z 325.454,A -85,B 0,C 180,E1 -18304.738,E2 -18304.738} C_VEL
LIN {X 0,Y 275.187,Z 309.432,A -85,B 0,C 180,E1 -18306.354,E2 -18306.354} C_VEL
LIN {X 0,Y 268.302,Z 296.615,A -85,B 0,C 180,E1 -18307.871,E2 -18307.871} C_VEL
LIN {X 0,Y 264.351,Z 289.591,A -85,B 0,C 180,E1 -18308.817,E2 -18308.817} C_VEL
LIN {X 0,Y 263.31,Z 286.197,A -85,B 0,C 180,E1 -18310.171,E2 -18310.171} C_VEL
LIN {X 0,Y 263.14,Z 285.328,A -85,B 0,C 180,E1 -18310.759,E2 -18310.759} C_VEL
LIN {X 0,Y 263.126,Z 285.316,A -85,B 0,C 180,E1 -18313.982,E2 -18313.982} C_VEL
LIN {X 0,Y 263.122,Z 285.29,A -85,B 0,C 180,E1 -18318.405,E2 -18318.405} C_VEL
LIN {X 0,Y 263.163,Z 285.334,A -85,B 0,C 180,E1 -18322.103,E2 -18322.103} C_VEL
LIN {X 0,Y 263.18,Z 285.273,A -85,B 0,C 180,E1 -18325.89,E2 -18325.89} C_VEL
LIN {X 0,Y 263.147,Z 285.313,A -85,B 0,C 180,E1 -18329.506,E2 -18329.506} C_VEL
LIN {X 0,Y 263.188,Z 285.313,A -85,B 0,C 180,E1 -18333.002,E2 -18333.002} C_VEL
LIN {X 0,Y 263.18,Z 285.328,A -85,B 0,C 180,E1 -18336.386,E2 -18336.386} C_VEL
LIN {X 0,Y 263.259,Z 285.299,A -85,B 0,C 180,E1 -18339.693,E2 -18339.693} C_VEL
LIN {X 0,Y 263.228,Z 285.315,A -85,B 0,C 180,E1 -18341.923,E2 -18341.923} C_VEL
LIN {X 0,Y 262.563,Z 285.398,A -85,B 0,C 180,E1 -18343.2,E2 -18343.2} C_VEL
LIN {X 0,Y 259.719,Z 285.747,A -85,B 0,C 180,E1 -18345.282,E2 -18345.282} C_VEL
LIN {X 0,Y 257.329,Z 286.049,A -85,B 0,C 180,E1 -18346.976,E2 -18346.976} C_VEL
LIN {X 0,Y 256.341,Z 286.179,A -85,B 0,C 180,E1 -18348.289,E2 -18348.289} C_VEL
LIN {X 0,Y 256.28,Z 286.181,A -85,B 0,C 180,E1 -18348.734,E2 -18348.734} C_VEL
LIN {X 0,Y 256.51,Z 286.139,A -85,B 0,C 180,E1 -18352.126,E2 -18352.126} C_VEL
LIN {X 0,Y 256.493,Z 286.137,A -85,B 0,C 180,E1 -18356.858,E2 -18356.858} C_VEL
LIN {X 0,Y 256.768,Z 286.122,A -85,B 0,C 180,E1 -18360,E2 -18360} C_VEL
LIN {X 0,Y 256.493,Z 286.14,A -85,B 0,C 180,E1 -18363.141,E2 -18363.141} C_VEL
LIN {X 0,Y 256.534,Z 286.153,A -85,B 0,C 180,E1 -18367.873,E2 -18367.873} C_VEL
LIN {X 0,Y 256.304,Z 286.163,A -85,B 0,C 180,E1 -18371.066,E2 -18371.066} C_VEL
LIN {X 0,Y 256.274,Z 286.168,A -85,B 0,C 180,E1 -18375.916,E2 -18375.916} C_VEL
LIN {X 0,Y 256.162,Z 286.19,A -85,B 0,C 180,E1 -18380.895,E2 -18380.895} C_VEL
LIN {X 0,Y 256.184,Z 286.199,A -85,B 0,C 180,E1 -18385.139,E2 -18385.139} C_VEL
LIN {X 0,Y 256.11,Z 286.208,A -85,B 0,C 180,E1 -18389.6,E2 -18389.6} C_VEL
LIN {X 0,Y 256.063,Z 286.16,A -85,B 0,C 180,E1 -18393.293,E2 -18393.293} C_VEL
LIN {X 0,Y 256.112,Z 286.188,A -85,B 0,C 180,E1 -18397.272,E2 -18397.272} C_VEL
LIN {X 0,Y 256.056,Z 286.205,A -85,B 0,C 180,E1 -18401.203,E2 -18401.203} C_VEL
LIN {X 0,Y 256.073,Z 286.214,A -85,B 0,C 180,E1 -18405.527,E2 -18405.527} C_VEL
LIN {X 0,Y 256.19,Z 286.423,A -85,B 0,C 180,E1 -18407.16,E2 -18407.16} C_VEL
LIN {X 0,Y 258.103,Z 292.998,A -85,B 0,C 180,E1 -18410.064,E2 -18410.064} C_VEL
LIN {X 0,Y 262.512,Z 301.056,A -85,B 0,C 180,E1 -18411.204,E2 -18411.204} C_VEL
LIN {X 0,Y 269.998,Z 315.377,A -85,B 0,C 180,E1 -18412.937,E2 -18412.937} C_VEL
LIN {X 0,Y 277.991,Z 332.859,A -85,B 0,C 180,E1 -18414.713,E2 -18414.713} C_VEL
LIN {X 0,Y 281.223,Z 341.017,A -85,B 0,C 180,E1 -18415.425,E2 -18415.425} C_VEL
LIN {X 0,Y 281.962,Z 346.093,A -85,B 0,C 180,E1 -18415.682,E2 -18415.682} C_VEL
LIN {X 0,Y 278.581,Z 429.535,A -85,B 0,C 180,E1 -18417.765,E2 -18417.765} C_VEL
LIN {X 0,Y 277.348,Z 443.575,A -85,B 0,C 180,E1 -18418.332,E2 -18418.332} C_VEL
LIN {X 0,Y 275.76,Z 456.88,A -85,B 0,C 180,E1 -18419.143,E2 -18419.143} C_VEL
LIN {X 0,Y 273.755,Z 469.502,A -85,B 0,C 180,E1 -18420.172,E2 -18420.172} C_VEL
LIN {X 0,Y 271.279,Z 482.626,A -85,B 0,C 180,E1 -18421.575,E2 -18421.575} C_VEL
LIN {X 0,Y 268.678,Z 494.861,A -85,B 0,C 180,E1 -18423.244,E2 -18423.244} C_VEL
LIN {X 0,Y 266.116,Z 505.341,A -85,B 0,C 180,E1 -18425.005,E2 -18425.005} C_VEL
LIN {X 0,Y 263.296,Z 516.061,A -85,B 0,C 180,E1 -18427.23,E2 -18427.23} C_VEL
LIN {X 0,Y 260.864,Z 524.912,A -85,B 0,C 180,E1 -18429.499,E2 -18429.499} C_VEL
LIN {X 0,Y 258.686,Z 533.311,A -85,B 0,C 180,E1 -18432.172,E2 -18432.172} C_VEL
LIN {X 0,Y 256.884,Z 540.233,A -85,B 0,C 180,E1 -18434.936,E2 -18434.936} C_VEL
LIN {X 0,Y 255.585,Z 544.942,A -85,B 0,C 180,E1 -18437.292,E2 -18437.292} C_VEL
LIN {X 0,Y 254.632,Z 549.825,A -85,B 0,C 180,E1 -18440.468,E2 -18440.468} C_VEL
LIN {X 0,Y 254.065,Z 553.219,A -85,B 0,C 180,E1 -18443.648,E2 -18443.648} C_VEL
LIN {X 0,Y 253.91,Z 555.225,A -85,B 0,C 180,E1 -18446.827,E2 -18446.827} C_VEL
LIN {X 0,Y 253.98,Z 555.886,A -85,B 0,C 180,E1 -18450,E2 -18450} C_VEL
LIN {X 0,Y 253.91,Z 555.211,A -85,B 0,C 180,E1 -18453.173,E2 -18453.173} C_VEL
LIN {X 0,Y 254.075,Z 553.192,A -85,B 0,C 180,E1 -18456.352,E2 -18456.352} C_VEL
LIN {X 0,Y 254.633,Z 549.783,A -85,B 0,C 180,E1 -18459.532,E2 -18459.532} C_VEL
LIN {X 0,Y 255.586,Z 544.879,A -85,B 0,C 180,E1 -18462.708,E2 -18462.708} C_VEL
LIN {X 0,Y 256.883,Z 540.153,A -85,B 0,C 180,E1 -18465.064,E2 -18465.064} C_VEL
LIN {X 0,Y 258.638,Z 532.752,A -85,B 0,C 180,E1 -18468,E2 -18468} C_VEL
LIN {X 0,Y 260.855,Z 524.792,A -85,B 0,C 180,E1 -18470.502,E2 -18470.502} C_VEL
LIN {X 0,Y 263.279,Z 515.916,A -85,B 0,C 180,E1 -18472.772,E2 -18472.772} C_VEL
LIN {X 0,Y 265.562,Z 507.118,A -85,B 0,C 180,E1 -18474.633,E2 -18474.633} C_VEL
LIN {X 0,Y 268.482,Z 495.63,A -85,B 0,C 180,E1 -18476.602,E2 -18476.602} C_VEL
LIN {X 0,Y 270.915,Z 484.079,A -85,B 0,C 180,E1 -18478.214,E2 -18478.214} C_VEL
LIN {X 0,Y 273.41,Z 470.946,A -85,B 0,C 180,E1 -18479.657,E2 -18479.657} C_VEL
LIN {X 0,Y 275.567,Z 457.587,A -85,B 0,C 180,E1 -18480.774,E2 -18480.774} C_VEL
LIN {X 0,Y 277.254,Z 443.781,A -85,B 0,C 180,E1 -18481.627,E2 -18481.627} C_VEL
LIN {X 0,Y 278.531,Z 429.916,A -85,B 0,C 180,E1 -18482.188,E2 -18482.188} C_VEL
LIN {X 0,Y 281.842,Z 345.594,A -85,B 0,C 180,E1 -18484.31,E2 -18484.31} C_VEL
LIN {X 0,Y 280.865,Z 339.914,A -85,B 0,C 180,E1 -18484.618,E2 -18484.618} C_VEL
LIN {X 0,Y 273.147,Z 321.918,A -85,B 0,C 180,E1 -18486.312,E2 -18486.312} C_VEL
LIN {X 0,Y 264.922,Z 305.567,A -85,B 0,C 180,E1 -18488.176,E2 -18488.176} C_VEL
LIN {X 0,Y 259.391,Z 295.78,A -85,B 0,C 180,E1 -18489.483,E2 -18489.483} C_VEL
LIN {X 0,Y 258.005,Z 292.928,A -85,B 0,C 180,E1 -18489.917,E2 -18489.917} C_VEL
LIN {X 0,Y 256.113,Z 286.366,A -85,B 0,C 180,E1 -18492.829,E2 -18492.829} C_VEL
LIN {X 0,Y 256.046,Z 286.21,A -85,B 0,C 180,E1 -18496.67,E2 -18496.67} C_VEL
LIN {X 0,Y 256.069,Z 286.211,A -85,B 0,C 180,E1 -18500.857,E2 -18500.857} C_VEL
LIN {X 0,Y 256.129,Z 286.179,A -85,B 0,C 180,E1 -18502.867,E2 -18502.867} C_VEL
LIN {X 0,Y 256.064,Z 286.16,A -85,B 0,C 180,E1 -18506.707,E2 -18506.707} C_VEL
LIN {X 0,Y 256.11,Z 286.207,A -85,B 0,C 180,E1 -18510.4,E2 -18510.4} C_VEL
LIN {X 0,Y 256.185,Z 286.199,A -85,B 0,C 180,E1 -18514.861,E2 -18514.861} C_VEL
LIN {X 0,Y 256.162,Z 286.191,A -85,B 0,C 180,E1 -18519.105,E2 -18519.105} C_VEL
LIN {X 0,Y 256.275,Z 286.168,A -85,B 0,C 180,E1 -18524.084,E2 -18524.084} C_VEL
LIN {X 0,Y 256.305,Z 286.163,A -85,B 0,C 180,E1 -18528.934,E2 -18528.934} C_VEL
LIN {X 0,Y 256.535,Z 286.153,A -85,B 0,C 180,E1 -18532.127,E2 -18532.127} C_VEL
LIN {X 0,Y 256.709,Z 286.131,A -85,B 0,C 180,E1 -18538.431,E2 -18538.431} C_VEL
LIN {X 0,Y 256.709,Z 286.111,A -85,B 0,C 180,E1 -18541.569,E2 -18541.569} C_VEL
LIN {X 0,Y 256.466,Z 286.155,A -85,B 0,C 180,E1 -18546.726,E2 -18546.726} C_VEL
LIN {X 0,Y 256.423,Z 286.147,A -85,B 0,C 180,E1 -18549.465,E2 -18549.465} C_VEL
LIN {X 0,Y 256.246,Z 286.171,A -85,B 0,C 180,E1 -18554.291,E2 -18554.291} C_VEL
LIN {X 0,Y 256.206,Z 286.196,A -85,B 0,C 180,E1 -18557.562,E2 -18557.562} C_VEL
LIN {X 0,Y 256.153,Z 286.183,A -85,B 0,C 180,E1 -18561.12,E2 -18561.12} C_VEL
LIN {X 0,Y 256.185,Z 286.187,A -85,B 0,C 180,E1 -18565.139,E2 -18565.139} C_VEL
LIN {X 0,Y 256.111,Z 286.205,A -85,B 0,C 180,E1 -18569.6,E2 -18569.6} C_VEL
LIN {X 0,Y 256.082,Z 286.149,A -85,B 0,C 180,E1 -18573.291,E2 -18573.291} C_VEL
LIN {X 0,Y 256.128,Z 286.204,A -85,B 0,C 180,E1 -18577.276,E2 -18577.276} C_VEL
LIN {X 0,Y 256.055,Z 286.168,A -85,B 0,C 180,E1 -18581.204,E2 -18581.204} C_VEL
LIN {X 0,Y 256.061,Z 286.206,A -85,B 0,C 180,E1 -18585.53,E2 -18585.53} C_VEL
LIN {X 0,Y 256.114,Z 286.37,A -85,B 0,C 180,E1 -18588.603,E2 -18588.603} C_VEL
LIN {X 0,Y 257.003,Z 289.495,A -85,B 0,C 180,E1 -18589.969,E2 -18589.969} C_VEL
LIN {X 0,Y 262.989,Z 299.935,A -85,B 0,C 180,E1 -18591.478,E2 -18591.478} C_VEL
LIN {X 0,Y 270.148,Z 313.281,A -85,B 0,C 180,E1 -18593.116,E2 -18593.116} C_VEL
LIN {X 0,Y 278.361,Z 330.961,A -85,B 0,C 180,E1 -18594.927,E2 -18594.927} C_VEL
LIN {X 0,Y 282.007,Z 339.929,A -85,B 0,C 180,E1 -18595.719,E2 -18595.719} C_VEL
LIN {X 0,Y 279.289,Z 410.306,A -85,B 0,C 180,E1 -18597.467,E2 -18597.467} C_VEL
LIN {X 0,Y 278.398,Z 428.724,A -85,B 0,C 180,E1 -18597.986,E2 -18597.986} C_VEL
LIN {X 0,Y 276.98,Z 443.286,A -85,B 0,C 180,E1 -18598.658,E2 -18598.658} C_VEL
LIN {X 0,Y 275.18,Z 457.181,A -85,B 0,C 180,E1 -18599.603,E2 -18599.603} C_VEL
LIN {X 0,Y 273.184,Z 469.641,A -85,B 0,C 180,E1 -18600.739,E2 -18600.739} C_VEL
LIN {X 0,Y 270.916,Z 481.852,A -85,B 0,C 180,E1 -18602.164,E2 -18602.164} C_VEL
LIN {X 0,Y 268.407,Z 493.042,A -85,B 0,C 180,E1 -18603.778,E2 -18603.778} C_VEL
LIN {X 0,Y 265.588,Z 504.292,A -85,B 0,C 180,E1 -18605.785,E2 -18605.785} C_VEL
LIN {X 0,Y 262.925,Z 514.344,A -85,B 0,C 180,E1 -18608.024,E2 -18608.024} C_VEL
LIN {X 0,Y 260.597,Z 522.689,A -85,B 0,C 180,E1 -18610.299,E2 -18610.299} C_VEL
LIN {X 0,Y 258.778,Z 529.652,A -85,B 0,C 180,E1 -18612.618,E2 -18612.618} C_VEL
LIN {X 0,Y 257.235,Z 535.398,A -85,B 0,C 180,E1 -18614.957,E2 -18614.957} C_VEL
LIN {X 0,Y 255.94,Z 540.121,A -85,B 0,C 180,E1 -18617.31,E2 -18617.31} C_VEL
LIN {X 0,Y 254.833,Z 545.012,A -85,B 0,C 180,E1 -18620.475,E2 -18620.475} C_VEL
LIN {X 0,Y 254.248,Z 548.414,A -85,B 0,C 180,E1 -18623.652,E2 -18623.652} C_VEL
LIN {X 0,Y 253.984,Z 550.433,A -85,B 0,C 180,E1 -18626.827,E2 -18626.827} C_VEL
LIN {X 0,Y 253.983,Z 551.121,A -85,B 0,C 180,E1 -18630,E2 -18630} C_VEL
LIN {X 0,Y 253.984,Z 550.49,A -85,B 0,C 180,E1 -18633.172,E2 -18633.172} C_VEL
LIN {X 0,Y 254.25,Z 548.523,A -85,B 0,C 180,E1 -18636.348,E2 -18636.348} C_VEL
LIN {X 0,Y 254.827,Z 545.174,A -85,B 0,C 180,E1 -18639.525,E2 -18639.525} C_VEL
LIN {X 0,Y 255.919,Z 540.343,A -85,B 0,C 180,E1 -18642.691,E2 -18642.691} C_VEL
LIN {X 0,Y 257.194,Z 535.679,A -85,B 0,C 180,E1 -18645.046,E2 -18645.046} C_VEL
LIN {X 0,Y 259.058,Z 528.689,A -85,B 0,C 180,E1 -18647.846,E2 -18647.846} C_VEL
LIN {X 0,Y 260.881,Z 521.823,A -85,B 0,C 180,E1 -18650.088,E2 -18650.088} C_VEL
LIN {X 0,Y 263.28,Z 513.301,A -85,B 0,C 180,E1 -18652.357,E2 -18652.357} C_VEL
LIN {X 0,Y 265.966,Z 502.972,A -85,B 0,C 180,E1 -18654.593,E2 -18654.593} C_VEL
LIN {X 0,Y 268.868,Z 491.416,A -85,B 0,C 180,E1 -18656.591,E2 -18656.591} C_VEL
LIN {X 0,Y 271.397,Z 479.554,A -85,B 0,C 180,E1 -18658.249,E2 -18658.249} C_VEL
LIN {X 0,Y 273.648,Z 467.187,A -85,B 0,C 180,E1 -18659.629,E2 -18659.629} C_VEL
LIN {X 0,Y 275.703,Z 454.05,A -85,B 0,C 180,E1 -18660.757,E2 -18660.757} C_VEL
LIN {X 0,Y 277.453,Z 439.817,A -85,B 0,C 180,E1 -18661.655,E2 -18661.655} C_VEL
LIN {X 0,Y 278.578,Z 426.266,A -85,B 0,C 180,E1 -18662.235,E2 -18662.235} C_VEL
LIN {X 0,Y 281.107,Z 367.55,A -85,B 0,C 180,E1 -18663.702,E2 -18663.702} C_VEL
LIN {X 0,Y 282.032,Z 339.947,A -85,B 0,C 180,E1 -18664.407,E2 -18664.407} C_VEL
LIN {X 0,Y 276.07,Z 325.697,A -85,B 0,C 180,E1 -18665.707,E2 -18665.707} C_VEL
LIN {X 0,Y 268.15,Z 309.4,A -85,B 0,C 180,E1 -18667.472,E2 -18667.472} C_VEL
LIN {X 0,Y 261.72,Z 297.695,A -85,B 0,C 180,E1 -18668.964,E2 -18668.964} C_VEL
LIN {X 0,Y 257.065,Z 289.624,A -85,B 0,C 180,E1 -18670.145,E2 -18670.145} C_VEL
LIN {X 0,Y 256.129,Z 286.414,A -85,B 0,C 180,E1 -18671.512,E2 -18671.512} C_VEL
LIN {X 0,Y 256.063,Z 286.187,A -85,B 0,C 180,E1 -18673.326,E2 -18673.326} C_VEL
LIN {X 0,Y 256.071,Z 286.171,A -85,B 0,C 180,E1 -18677.818,E2 -18677.818} C_VEL
LIN {X 0,Y 256.085,Z 286.191,A -85,B 0,C 180,E1 -18680.86,E2 -18680.86} C_VEL
LIN {X 0,Y 256.117,Z 286.166,A -85,B 0,C 180,E1 -18684.812,E2 -18684.812} C_VEL
LIN {X 0,Y 256.088,Z 286.169,A -85,B 0,C 180,E1 -18688.572,E2 -18688.572} C_VEL
LIN {X 0,Y 256.138,Z 286.202,A -85,B 0,C 180,E1 -18692.196,E2 -18692.196} C_VEL
LIN {X 0,Y 256.163,Z 286.199,A -85,B 0,C 180,E1 -18695.699,E2 -18695.699} C_VEL
LIN {X 0,Y 256.162,Z 286.182,A -85,B 0,C 180,E1 -18699.104,E2 -18699.104} C_VEL
LIN {X 0,Y 256.289,Z 286.168,A -85,B 0,C 180,E1 -18704.084,E2 -18704.084} C_VEL
LIN {X 0,Y 256.28,Z 286.181,A -85,B 0,C 180,E1 -18708.734,E2 -18708.734} C_VEL
LIN {X 0,Y 255.655,Z 286.266,A -85,B 0,C 180,E1 -18710.048,E2 -18710.048} C_VEL
LIN {X 0,Y 252.793,Z 286.63,A -85,B 0,C 180,E1 -18712.19,E2 -18712.19} C_VEL
LIN {X 0,Y 250.368,Z 286.928,A -85,B 0,C 180,E1 -18713.934,E2 -18713.934} C_VEL
LIN {X 0,Y 249.374,Z 287.043,A -85,B 0,C 180,E1 -18715.287,E2 -18715.287} C_VEL
LIN {X 0,Y 249.32,Z 287.04,A -85,B 0,C 180,E1 -18715.745,E2 -18715.745} C_VEL
LIN {X 0,Y 249.671,Z 286.986,A -85,B 0,C 180,E1 -18718.387,E2 -18718.387} C_VEL
LIN {X 0,Y 249.671,Z 287.008,A -85,B 0,C 180,E1 -18721.613,E2 -18721.613} C_VEL
LIN {X 0,Y 249.455,Z 287.033,A -85,B 0,C 180,E1 -18726.47,E2 -18726.47} C_VEL
LIN {X 0,Y 249.384,Z 287.024,A -85,B 0,C 180,E1 -18729.735,E2 -18729.735} C_VEL
LIN {X 0,Y 249.192,Z 287.062,A -85,B 0,C 180,E1 -18734.704,E2 -18734.704} C_VEL
LIN {X 0,Y 249.13,Z 287.068,A -85,B 0,C 180,E1 -18738.078,E2 -18738.078} C_VEL
LIN {X 0,Y 249.082,Z 287.066,A -85,B 0,C 180,E1 -18741.518,E2 -18741.518} C_VEL
LIN {X 0,Y 249.126,Z 287.076,A -85,B 0,C 180,E1 -18745.482,E2 -18745.482} C_VEL
LIN {X 0,Y 249.079,Z 287.078,A -85,B 0,C 180,E1 -18748.994,E2 -18748.994} C_VEL
LIN {X 0,Y 249.026,Z 287.048,A -85,B 0,C 180,E1 -18752.426,E2 -18752.426} C_VEL
LIN {X 0,Y 249.027,Z 287.047,A -85,B 0,C 180,E1 -18756.346,E2 -18756.346} C_VEL
LIN {X 0,Y 249.004,Z 287.081,A -85,B 0,C 180,E1 -18760.478,E2 -18760.478} C_VEL
LIN {X 0,Y 249.016,Z 287.086,A -85,B 0,C 180,E1 -18764.876,E2 -18764.876} C_VEL
LIN {X 0,Y 249.084,Z 287.367,A -85,B 0,C 180,E1 -18766.073,E2 -18766.073} C_VEL
LIN {X 0,Y 250.794,Z 292.952,A -85,B 0,C 180,E1 -18768.657,E2 -18768.657} C_VEL
LIN {X 0,Y 256.838,Z 303.605,A -85,B 0,C 180,E1 -18770.272,E2 -18770.272} C_VEL
LIN {X 0,Y 264.859,Z 318.915,A -85,B 0,C 180,E1 -18772.213,E2 -18772.213} C_VEL
LIN {X 0,Y 272.479,Z 335.764,A -85,B 0,C 180,E1 -18773.983,E2 -18773.983} C_VEL
LIN {X 0,Y 275.584,Z 343.538,A -85,B 0,C 180,E1 -18774.693,E2 -18774.693} C_VEL
LIN {X 0,Y 276.059,Z 347.482,A -85,B 0,C 180,E1 -18774.886,E2 -18774.886} C_VEL
LIN {X 0,Y 272.595,Z 429.759,A -85,B 0,C 180,E1 -18776.978,E2 -18776.978} C_VEL
LIN {X 0,Y 271.245,Z 444.307,A -85,B 0,C 180,E1 -18777.588,E2 -18777.588} C_VEL
LIN {X 0,Y 269.693,Z 456.82,A -85,B 0,C 180,E1 -18778.37,E2 -18778.37} C_VEL
LIN {X 0,Y 267.609,Z 469.44,A -85,B 0,C 180,E1 -18779.415,E2 -18779.415} C_VEL
LIN {X 0,Y 265.034,Z 482.558,A -85,B 0,C 180,E1 -18780.84,E2 -18780.84} C_VEL
LIN {X 0,Y 262.301,Z 494.957,A -85,B 0,C 180,E1 -18782.569,E2 -18782.569} C_VEL
LIN {X 0,Y 259.679,Z 505.277,A -85,B 0,C 180,E1 -18784.341,E2 -18784.341} C_VEL
LIN {X 0,Y 256.745,Z 515.997,A -85,B 0,C 180,E1 -18786.615,E2 -18786.615} C_VEL
LIN {X 0,Y 254.177,Z 524.847,A -85,B 0,C 180,E1 -18788.934,E2 -18788.934} C_VEL
LIN {X 0,Y 251.895,Z 532.921,A -85,B 0,C 180,E1 -18791.553,E2 -18791.553} C_VEL
LIN {X 0,Y 249.994,Z 540.168,A -85,B 0,C 180,E1 -18794.51,E2 -18794.51} C_VEL
LIN {X 0,Y 248.621,Z 544.876,A -85,B 0,C 180,E1 -18796.93,E2 -18796.93} C_VEL
LIN {X 0,Y 247.598,Z 549.759,A -85,B 0,C 180,E1 -18800.195,E2 -18800.195} C_VEL
LIN {X 0,Y 247.009,Z 553.153,A -85,B 0,C 180,E1 -18803.465,E2 -18803.465} C_VEL
LIN {X 0,Y 246.817,Z 555.159,A -85,B 0,C 180,E1 -18806.735,E2 -18806.735} C_VEL
LIN {X 0,Y 246.89,Z 555.819,A -85,B 0,C 180,E1 -18810,E2 -18810} C_VEL
LIN {X 0,Y 246.817,Z 555.144,A -85,B 0,C 180,E1 -18813.265,E2 -18813.265} C_VEL
LIN {X 0,Y 247.015,Z 553.125,A -85,B 0,C 180,E1 -18816.535,E2 -18816.535} C_VEL
LIN {X 0,Y 247.6,Z 549.715,A -85,B 0,C 180,E1 -18819.806,E2 -18819.806} C_VEL
LIN {X 0,Y 248.622,Z 544.811,A -85,B 0,C 180,E1 -18823.07,E2 -18823.07} C_VEL
LIN {X 0,Y 249.992,Z 540.085,A -85,B 0,C 180,E1 -18825.49,E2 -18825.49} C_VEL
LIN {X 0,Y 251.738,Z 533.138,A -85,B 0,C 180,E1 -18828.339,E2 -18828.339} C_VEL
LIN {X 0,Y 254.169,Z 524.723,A -85,B 0,C 180,E1 -18831.067,E2 -18831.067} C_VEL
LIN {X 0,Y 256.727,Z 515.847,A -85,B 0,C 180,E1 -18833.387,E2 -18833.387} C_VEL
LIN {X 0,Y 259.122,Z 507.048,A -85,B 0,C 180,E1 -18835.288,E2 -18835.288} C_VEL
LIN {X 0,Y 261.906,Z 496.561,A -85,B 0,C 180,E1 -18837.14,E2 -18837.14} C_VEL
LIN {X 0,Y 264.438,Z 485.147,A -85,B 0,C 180,E1 -18838.797,E2 -18838.797} C_VEL
LIN {X 0,Y 266.93,Z 472.642,A -85,B 0,C 180,E1 -18840.234,E2 -18840.234} C_VEL
LIN {X 0,Y 269.303,Z 458.644,A -85,B 0,C 180,E1 -18841.462,E2 -18841.462} C_VEL
LIN {X 0,Y 271.157,Z 444.479,A -85,B 0,C 180,E1 -18842.369,E2 -18842.369} C_VEL
LIN {X 0,Y 272.454,Z 431.091,A -85,B 0,C 180,E1 -18842.941,E2 -18842.941} C_VEL
LIN {X 0,Y 275.739,Z 352.421,A -85,B 0,C 180,E1 -18844.964,E2 -18844.964} C_VEL
LIN {X 0,Y 275.901,Z 345.952,A -85,B 0,C 180,E1 -18845.142,E2 -18845.142} C_VEL
LIN {X 0,Y 275.085,Z 342.202,A -85,B 0,C 180,E1 -18845.379,E2 -18845.379} C_VEL
LIN {X 0,Y 267.719,Z 325.026,A -85,B 0,C 180,E1 -18847.065,E2 -18847.065} C_VEL
LIN {X 0,Y 260.193,Z 309.859,A -85,B 0,C 180,E1 -18848.848,E2 -18848.848} C_VEL
LIN {X 0,Y 253.026,Z 297.052,A -85,B 0,C 180,E1 -18850.63,E2 -18850.63} C_VEL
LIN {X 0,Y 250.69,Z 292.846,A -85,B 0,C 180,E1 -18851.326,E2 -18851.326} C_VEL
LIN {X 0,Y 249.064,Z 287.271,A -85,B 0,C 180,E1 -18853.928,E2 -18853.928} C_VEL
LIN {X 0,Y 249.007,Z 287.094,A -85,B 0,C 180,E1 -18857.361,E2 -18857.361} C_VEL
LIN {X 0,Y 249.023,Z 287.091,A -85,B 0,C 180,E1 -18861.619,E2 -18861.619} C_VEL
LIN {X 0,Y 249.04,Z 287.027,A -85,B 0,C 180,E1 -18865.639,E2 -18865.639} C_VEL
LIN {X 0,Y 249.048,Z 287.086,A -85,B 0,C 180,E1 -18869.473,E2 -18869.473} C_VEL
LIN {X 0,Y 249.07,Z 287.069,A -85,B 0,C 180,E1 -18873.162,E2 -18873.162} C_VEL
LIN {X 0,Y 249.075,Z 287.07,A -85,B 0,C 180,E1 -18876.732,E2 -18876.732} C_VEL
LIN {X 0,Y 249.107,Z 287.08,A -85,B 0,C 180,E1 -18880.211,E2 -18880.211} C_VEL
LIN {X 0,Y 249.219,Z 287.045,A -85,B 0,C 180,E1 -18883.62,E2 -18883.62} C_VEL
LIN {X 0,Y 249.248,Z 287.044,A -85,B 0,C 180,E1 -18888.616,E2 -18888.616} C_VEL
LIN {X 0,Y 249.477,Z 287.029,A -85,B 0,C 180,E1 -18891.903,E2 -18891.903} C_VEL
LIN {X 0,Y 249.43,Z 287.018,A -85,B 0,C 180,E1 -18896.77,E2 -18896.77} C_VEL
LIN {X 0,Y 249.723,Z 287,A -85,B 0,C 180,E1 -18900,E2 -18900} C_VEL
LIN {X 0,Y 249.431,Z 287.016,A -85,B 0,C 180,E1 -18903.231,E2 -18903.231} C_VEL
LIN {X 0,Y 249.436,Z 287.033,A -85,B 0,C 180,E1 -18906.711,E2 -18906.711} C_VEL
LIN {X 0,Y 249.339,Z 287.03,A -85,B 0,C 180,E1 -18909.737,E2 -18909.737} C_VEL
LIN {X 0,Y 249.196,Z 287.047,A -85,B 0,C 180,E1 -18914.704,E2 -18914.704} C_VEL
LIN {X 0,Y 249.135,Z 287.077,A -85,B 0,C 180,E1 -18918.078,E2 -18918.078} C_VEL
LIN {X 0,Y 249.084,Z 287.065,A -85,B 0,C 180,E1 -18921.519,E2 -18921.519} C_VEL
LIN {X 0,Y 249.127,Z 287.062,A -85,B 0,C 180,E1 -18925.483,E2 -18925.483} C_VEL
LIN {X 0,Y 249.081,Z 287.085,A -85,B 0,C 180,E1 -18928.994,E2 -18928.994} C_VEL
LIN {X 0,Y 249.033,Z 287.031,A -85,B 0,C 180,E1 -18932.426,E2 -18932.426} C_VEL
LIN {X 0,Y 249.068,Z 287.06,A -85,B 0,C 180,E1 -18936.339,E2 -18936.339} C_VEL
LIN {X 0,Y 249.024,Z 287.048,A -85,B 0,C 180,E1 -18940.475,E2 -18940.475} C_VEL
LIN {X 0,Y 249.007,Z 287.094,A -85,B 0,C 180,E1 -18944.879,E2 -18944.879} C_VEL
LIN {X 0,Y 249.052,Z 287.277,A -85,B 0,C 180,E1 -18947.517,E2 -18947.517} C_VEL
LIN {X 0,Y 249.822,Z 289.713,A -85,B 0,C 180,E1 -18948.59,E2 -18948.59} C_VEL
LIN {X 0,Y 258.076,Z 303.835,A -85,B 0,C 180,E1 -18950.739,E2 -18950.739} C_VEL
LIN {X 0,Y 265.527,Z 317.966,A -85,B 0,C 180,E1 -18952.519,E2 -18952.519} C_VEL
LIN {X 0,Y 273.057,Z 334.408,A -85,B 0,C 180,E1 -18954.249,E2 -18954.249} C_VEL
LIN {X 0,Y 276.1,Z 341.789,A -85,B 0,C 180,E1 -18954.934,E2 -18954.934} C_VEL
LIN {X 0,Y 273.119,Z 415.635,A -85,B 0,C 180,E1 -18956.799,E2 -18956.799} C_VEL
LIN {X 0,Y 272.23,Z 431.083,A -85,B 0,C 180,E1 -18957.281,E2 -18957.281} C_VEL
LIN {X 0,Y 270.812,Z 444.885,A -85,B 0,C 180,E1 -18957.969,E2 -18957.969} C_VEL
LIN {X 0,Y 268.911,Z 458.378,A -85,B 0,C 180,E1 -18958.925,E2 -18958.925} C_VEL
LIN {X 0,Y 266.731,Z 471.302,A -85,B 0,C 180,E1 -18960.161,E2 -18960.161} C_VEL
LIN {X 0,Y 264.359,Z 483.282,A -85,B 0,C 180,E1 -18961.628,E2 -18961.628} C_VEL
LIN {X 0,Y 261.497,Z 495.303,A -85,B 0,C 180,E1 -18963.461,E2 -18963.461} C_VEL
LIN {X 0,Y 258.623,Z 506.141,A -85,B 0,C 180,E1 -18965.518,E2 -18965.518} C_VEL
LIN {X 0,Y 255.898,Z 515.896,A -85,B 0,C 180,E1 -18967.813,E2 -18967.813} C_VEL
LIN {X 0,Y 253.517,Z 523.987,A -85,B 0,C 180,E1 -18970.148,E2 -18970.148} C_VEL
LIN {X 0,Y 251.509,Z 531.731,A -85,B 0,C 180,E1 -18972.938,E2 -18972.938} C_VEL
LIN {X 0,Y 249.82,Z 537.142,A -85,B 0,C 180,E1 -18975.334,E2 -18975.334} C_VEL
LIN {X 0,Y 248.358,Z 542.828,A -85,B 0,C 180,E1 -18978.575,E2 -18978.575} C_VEL
LIN {X 0,Y 247.44,Z 546.959,A -85,B 0,C 180,E1 -18981.836,E2 -18981.836} C_VEL
LIN {X 0,Y 246.991,Z 549.659,A -85,B 0,C 180,E1 -18985.103,E2 -18985.103} C_VEL
LIN {X 0,Y 246.877,Z 551.009,A -85,B 0,C 180,E1 -18988.369,E2 -18988.369} C_VEL
LIN {X 0,Y 246.893,Z 551.188,A -85,B 0,C 180,E1 -18990,E2 -18990} C_VEL
LIN {X 0,Y 246.89,Z 550.557,A -85,B 0,C 180,E1 -18993.264,E2 -18993.264} C_VEL
LIN {X 0,Y 247.18,Z 548.589,A -85,B 0,C 180,E1 -18996.53,E2 -18996.53} C_VEL
